REGION Network 14: LH Thermocouple | IW 308
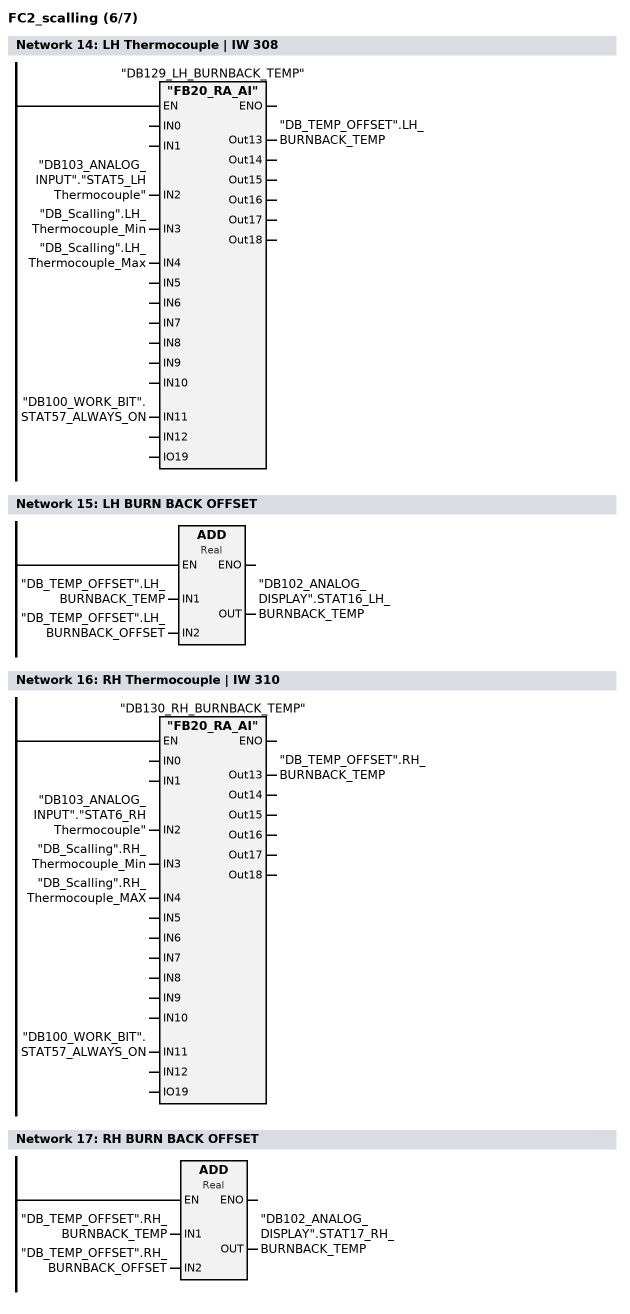
   RUNG wire#powerrail
      "DB129_LH_BURNBACK_TEMP"(IN0 :=, IN1 :=, IN2 := "DB103_ANALOG_INPUT"."STAT5_LH Thermocouple", IN3 := "DB_Scalling".LH_Thermocouple_Min, IN4 := "DB_Scalling".LH_Thermocouple_Max, IN5 :=, IN6 :=, IN7 :=, IN8 :=, IN9 :=, IN10 :=, IN11 := "DB100_WORK_BIT".STAT57_ALWAYS_ON, IN12 :=, IO19 :=, Out13 => "DB_TEMP_OFFSET".LH_BURNBACK_TEMP, Out14 =>, Out15 =>, Out16 =>, Out17 =>, Out18 =>)
   END_RUNG
   // the same network as SCL:
   "DB129_LH_BURNBACK_TEMP"(IN2 := "DB103_ANALOG_INPUT"."STAT5_LH Thermocouple",   // "FB20_RA_AI"
                           IN3 := "DB_Scalling".LH_Thermocouple_Min,
                           IN4 := "DB_Scalling".LH_Thermocouple_Max,
                           IN11 := "DB100_WORK_BIT".STAT57_ALWAYS_ON,
                           Out13 => "DB_TEMP_OFFSET".LH_BURNBACK_TEMP);
END_REGION

REGION Network 15: LH BURN BACK OFFSET
   RUNG wire#powerrail
      { S7_Templates := "SrcType := Real" } Add(in1 := "DB_TEMP_OFFSET".LH_BURNBACK_TEMP, in2 := "DB_TEMP_OFFSET".LH_BURNBACK_OFFSET, out => "DB102_ANALOG_DISPLAY".STAT16_LH_BURNBACK_TEMP)
   END_RUNG
   // the same network as SCL:
   "DB102_ANALOG_DISPLAY".STAT16_LH_BURNBACK_TEMP := "DB_TEMP_OFFSET".LH_BURNBACK_TEMP + "DB_TEMP_OFFSET".LH_BURNBACK_OFFSET;
END_REGION

REGION Network 16: RH Thermocouple | IW 310
   RUNG wire#powerrail
      "DB130_RH_BURNBACK_TEMP"(IN0 :=, IN1 :=, IN2 := "DB103_ANALOG_INPUT"."STAT6_RH Thermocouple", IN3 := "DB_Scalling".RH_Thermocouple_Min, IN4 := "DB_Scalling".RH_Thermocouple_MAX, IN5 :=, IN6 :=, IN7 :=, IN8 :=, IN9 :=, IN10 :=, IN11 := "DB100_WORK_BIT".STAT57_ALWAYS_ON, IN12 :=, IO19 :=, Out13 => "DB_TEMP_OFFSET".RH_BURNBACK_TEMP, Out14 =>, Out15 =>, Out16 =>, Out17 =>, Out18 =>)
   END_RUNG
   // the same network as SCL:
   "DB130_RH_BURNBACK_TEMP"(IN2 := "DB103_ANALOG_INPUT"."STAT6_RH Thermocouple",   // "FB20_RA_AI"
                           IN3 := "DB_Scalling".RH_Thermocouple_Min,
                           IN4 := "DB_Scalling".RH_Thermocouple_MAX,
                           IN11 := "DB100_WORK_BIT".STAT57_ALWAYS_ON,
                           Out13 => "DB_TEMP_OFFSET".RH_BURNBACK_TEMP);
END_REGION

REGION Network 17: RH BURN BACK OFFSET
   RUNG wire#powerrail
      { S7_Templates := "SrcType := Real" } Add(in1 := "DB_TEMP_OFFSET".RH_BURNBACK_TEMP, in2 := "DB_TEMP_OFFSET".RH_BURNBACK_OFFSET, out => "DB102_ANALOG_DISPLAY".STAT17_RH_BURNBACK_TEMP)
   END_RUNG
   // the same network as SCL:
   "DB102_ANALOG_DISPLAY".STAT17_RH_BURNBACK_TEMP := "DB_TEMP_OFFSET".RH_BURNBACK_TEMP + "DB_TEMP_OFFSET".RH_BURNBACK_OFFSET;
END_REGION

REGION Network 18: Poti LH Rear Undgrt | IW 304
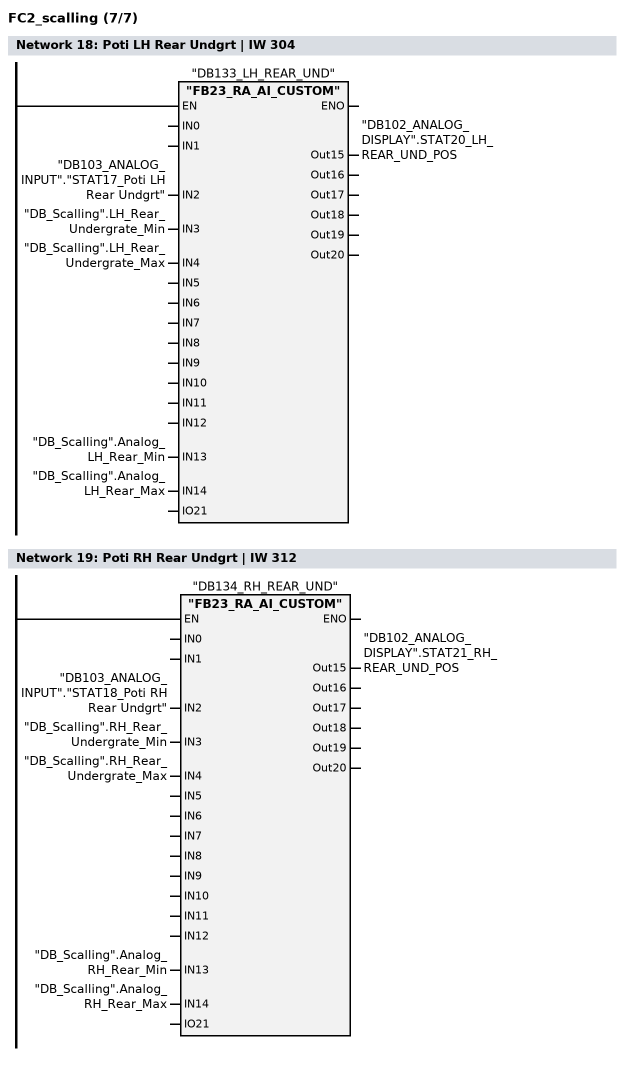
   RUNG wire#powerrail
      "DB133_LH_REAR_UND"(IN0 :=, IN1 :=, IN2 := "DB103_ANALOG_INPUT"."STAT17_Poti LH Rear Undgrt", IN3 := "DB_Scalling".LH_Rear_Undergrate_Min, IN4 := "DB_Scalling".LH_Rear_Undergrate_Max, IN5 :=, IN6 :=, IN7 :=, IN8 :=, IN9 :=, IN10 :=, IN11 :=, IN12 :=, IN13 := "DB_Scalling".Analog_LH_Rear_Min, IN14 := "DB_Scalling".Analog_LH_Rear_Max, IO21 :=, Out15 => "DB102_ANALOG_DISPLAY".STAT20_LH_REAR_UND_POS, Out16 =>, Out17 =>, Out18 =>, Out19 =>, Out20 =>)
   END_RUNG
   // the same network as SCL:
   "DB133_LH_REAR_UND"(IN2 := "DB103_ANALOG_INPUT"."STAT17_Poti LH Rear Undgrt",   // "FB23_RA_AI_CUSTOM"
                       IN3 := "DB_Scalling".LH_Rear_Undergrate_Min,
                       IN4 := "DB_Scalling".LH_Rear_Undergrate_Max,
                       IN13 := "DB_Scalling".Analog_LH_Rear_Min,
                       IN14 := "DB_Scalling".Analog_LH_Rear_Max,
                       Out15 => "DB102_ANALOG_DISPLAY".STAT20_LH_REAR_UND_POS);
END_REGION

REGION Network 19: Poti RH Rear Undgrt | IW 312
   RUNG wire#powerrail
      "DB134_RH_REAR_UND"(IN0 :=, IN1 :=, IN2 := "DB103_ANALOG_INPUT"."STAT18_Poti RH Rear Undgrt", IN3 := "DB_Scalling".RH_Rear_Undergrate_Min, IN4 := "DB_Scalling".RH_Rear_Undergrate_Max, IN5 :=, IN6 :=, IN7 :=, IN8 :=, IN9 :=, IN10 :=, IN11 :=, IN12 :=, IN13 := "DB_Scalling".Analog_RH_Rear_Min, IN14 := "DB_Scalling".Analog_RH_Rear_Max, IO21 :=, Out15 => "DB102_ANALOG_DISPLAY".STAT21_RH_REAR_UND_POS, Out16 =>, Out17 =>, Out18 =>, Out19 =>, Out20 =>)
   END_RUNG
   // the same network as SCL:
   "DB134_RH_REAR_UND"(IN2 := "DB103_ANALOG_INPUT"."STAT18_Poti RH Rear Undgrt",   // "FB23_RA_AI_CUSTOM"
                       IN3 := "DB_Scalling".RH_Rear_Undergrate_Min,
                       IN4 := "DB_Scalling".RH_Rear_Undergrate_Max,
                       IN13 := "DB_Scalling".Analog_RH_Rear_Min,
                       IN14 := "DB_Scalling".Analog_RH_Rear_Max,
                       Out15 => "DB102_ANALOG_DISPLAY".STAT21_RH_REAR_UND_POS);
END_REGION
END_FUNCTION

FUNCTION "FC3_BOILER_OPERATION" : Void   // FC3, LAD
TITLE = BOILER OPERATION
{ S7_Optimized_Access := 'TRUE' }
VERSION : 0.1
BEGIN

REGION Network 1: Ready For Operation ==> I 0.1
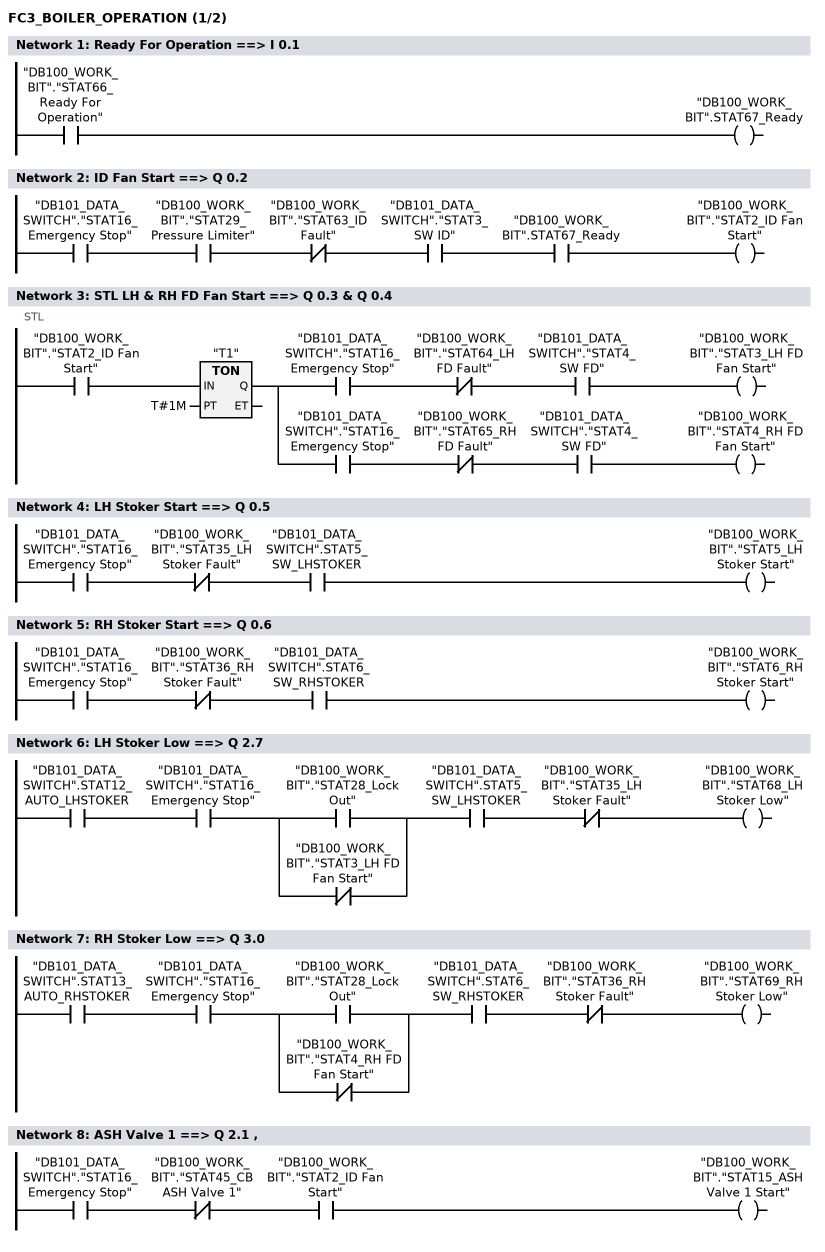
   RUNG wire#powerrail
      Contact( "DB100_WORK_BIT"."STAT66_Ready For Operation" )
      Coil( "DB100_WORK_BIT".STAT67_Ready )
   END_RUNG
   // the same network as SCL:
   "DB100_WORK_BIT".STAT67_Ready := "DB100_WORK_BIT"."STAT66_Ready For Operation";
END_REGION

REGION Network 2: ID Fan Start ==> Q 0.2
   RUNG wire#powerrail
      Contact( "DB101_DATA_SWITCH"."STAT16_Emergency Stop" )
      Contact( "DB100_WORK_BIT"."STAT29_Pressure Limiter" )
      I_Contact( "DB100_WORK_BIT"."STAT63_ID Fault" )
      Contact( "DB101_DATA_SWITCH"."STAT3_SW ID" )
      Contact( "DB100_WORK_BIT".STAT67_Ready )
      Coil( "DB100_WORK_BIT"."STAT2_ID Fan Start" )
   END_RUNG
   // the same network as SCL:
   "DB100_WORK_BIT"."STAT2_ID Fan Start" := "DB101_DATA_SWITCH"."STAT16_Emergency Stop" AND "DB100_WORK_BIT"."STAT29_Pressure Limiter" AND NOT "DB100_WORK_BIT"."STAT63_ID Fault" AND "DB101_DATA_SWITCH"."STAT3_SW ID" AND "DB100_WORK_BIT".STAT67_Ready;
END_REGION

REGION Network 3: STL LH & RH FD Fan Start ==> Q 0.3 & Q 0.4
   // STL
   "T1".TON(IN := "DB100_WORK_BIT"."STAT2_ID Fan Start", PT := T#1M);
   "DB100_WORK_BIT"."STAT3_LH FD Fan Start" := "T1".Q AND "DB101_DATA_SWITCH"."STAT16_Emergency Stop" AND NOT "DB100_WORK_BIT"."STAT64_LH FD Fault" AND "DB101_DATA_SWITCH"."STAT4_SW FD";
   "DB100_WORK_BIT"."STAT4_RH FD Fan Start" := "T1".Q AND "DB101_DATA_SWITCH"."STAT16_Emergency Stop" AND NOT "DB100_WORK_BIT"."STAT65_RH FD Fault" AND "DB101_DATA_SWITCH"."STAT4_SW FD";
END_REGION

REGION Network 4: LH Stoker Start ==> Q 0.5
   RUNG wire#powerrail
      Contact( "DB101_DATA_SWITCH"."STAT16_Emergency Stop" )
      I_Contact( "DB100_WORK_BIT"."STAT35_LH Stoker Fault" )
      Contact( "DB101_DATA_SWITCH".STAT5_SW_LHSTOKER )
      Coil( "DB100_WORK_BIT"."STAT5_LH Stoker Start" )
   END_RUNG
   // the same network as SCL:
   "DB100_WORK_BIT"."STAT5_LH Stoker Start" := "DB101_DATA_SWITCH"."STAT16_Emergency Stop" AND NOT "DB100_WORK_BIT"."STAT35_LH Stoker Fault" AND "DB101_DATA_SWITCH".STAT5_SW_LHSTOKER;
END_REGION

REGION Network 5: RH Stoker Start ==> Q 0.6
   RUNG wire#powerrail
      Contact( "DB101_DATA_SWITCH"."STAT16_Emergency Stop" )
      I_Contact( "DB100_WORK_BIT"."STAT36_RH Stoker Fault" )
      Contact( "DB101_DATA_SWITCH".STAT6_SW_RHSTOKER )
      Coil( "DB100_WORK_BIT"."STAT6_RH Stoker Start" )
   END_RUNG
   // the same network as SCL:
   "DB100_WORK_BIT"."STAT6_RH Stoker Start" := "DB101_DATA_SWITCH"."STAT16_Emergency Stop" AND NOT "DB100_WORK_BIT"."STAT36_RH Stoker Fault" AND "DB101_DATA_SWITCH".STAT6_SW_RHSTOKER;
END_REGION

REGION Network 6: LH Stoker Low ==> Q 2.7
   RUNG wire#powerrail
      Contact( "DB101_DATA_SWITCH".STAT12_AUTO_LHSTOKER )
      Contact( "DB101_DATA_SWITCH"."STAT16_Emergency Stop" )
      wire#w1
      Contact( "DB100_WORK_BIT"."STAT28_Lock Out" )
      wire#w2
      Contact( "DB101_DATA_SWITCH".STAT5_SW_LHSTOKER )
      I_Contact( "DB100_WORK_BIT"."STAT35_LH Stoker Fault" )
      Coil( "DB100_WORK_BIT"."STAT68_LH Stoker Low" )
   END_RUNG
   RUNG wire#w1
      I_Contact( "DB100_WORK_BIT"."STAT3_LH FD Fan Start" )
   END_RUNG wire#w2
   // the same network as SCL:
   "DB100_WORK_BIT"."STAT68_LH Stoker Low" := "DB101_DATA_SWITCH".STAT12_AUTO_LHSTOKER AND "DB101_DATA_SWITCH"."STAT16_Emergency Stop" AND ("DB100_WORK_BIT"."STAT28_Lock Out" OR NOT "DB100_WORK_BIT"."STAT3_LH FD Fan Start") AND "DB101_DATA_SWITCH".STAT5_SW_LHSTOKER AND NOT "DB100_WORK_BIT"."STAT35_LH Stoker Fault";
END_REGION

REGION Network 7: RH Stoker Low ==> Q 3.0
   RUNG wire#powerrail
      Contact( "DB101_DATA_SWITCH".STAT13_AUTO_RHSTOKER )
      Contact( "DB101_DATA_SWITCH"."STAT16_Emergency Stop" )
      wire#w1
      Contact( "DB100_WORK_BIT"."STAT28_Lock Out" )
      wire#w2
      Contact( "DB101_DATA_SWITCH".STAT6_SW_RHSTOKER )
      I_Contact( "DB100_WORK_BIT"."STAT36_RH Stoker Fault" )
      Coil( "DB100_WORK_BIT"."STAT69_RH Stoker Low" )
   END_RUNG
   RUNG wire#w1
      I_Contact( "DB100_WORK_BIT"."STAT4_RH FD Fan Start" )
   END_RUNG wire#w2
   // the same network as SCL:
   "DB100_WORK_BIT"."STAT69_RH Stoker Low" := "DB101_DATA_SWITCH".STAT13_AUTO_RHSTOKER AND "DB101_DATA_SWITCH"."STAT16_Emergency Stop" AND ("DB100_WORK_BIT"."STAT28_Lock Out" OR NOT "DB100_WORK_BIT"."STAT4_RH FD Fan Start") AND "DB101_DATA_SWITCH".STAT6_SW_RHSTOKER AND NOT "DB100_WORK_BIT"."STAT36_RH Stoker Fault";
END_REGION

REGION Network 8: ASH Valve 1 ==> Q 2.1 ,
   RUNG wire#powerrail
      Contact( "DB101_DATA_SWITCH"."STAT16_Emergency Stop" )
      I_Contact( "DB100_WORK_BIT"."STAT45_CB ASH Valve 1" )
      Contact( "DB100_WORK_BIT"."STAT2_ID Fan Start" )
      Coil( "DB100_WORK_BIT"."STAT15_ASH Valve 1 Start" )
   END_RUNG
   // the same network as SCL:
   "DB100_WORK_BIT"."STAT15_ASH Valve 1 Start" := "DB101_DATA_SWITCH"."STAT16_Emergency Stop" AND NOT "DB100_WORK_BIT"."STAT45_CB ASH Valve 1" AND "DB100_WORK_BIT"."STAT2_ID Fan Start";
END_REGION

REGION Network 9: ASH Valve 2 ==> Q 2.2
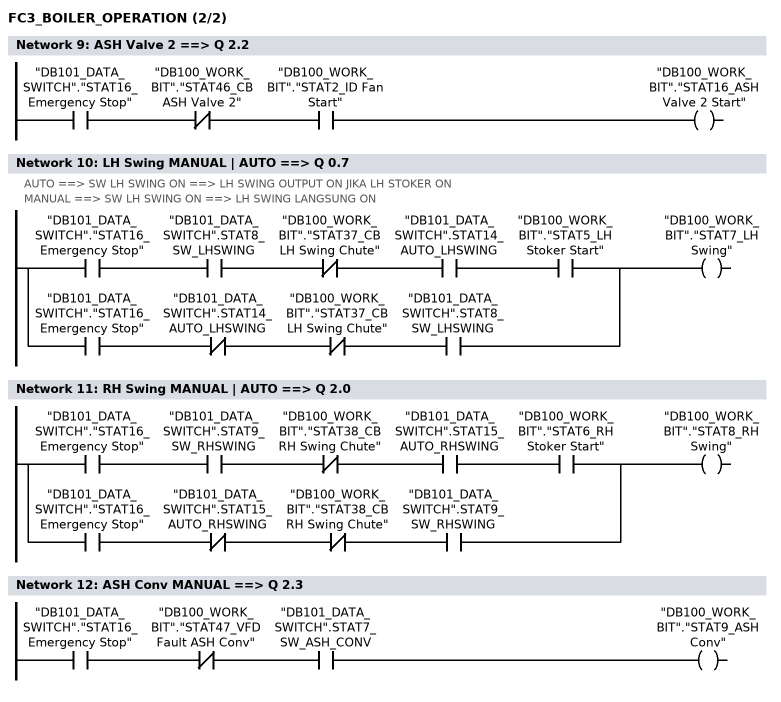
   RUNG wire#powerrail
      Contact( "DB101_DATA_SWITCH"."STAT16_Emergency Stop" )
      I_Contact( "DB100_WORK_BIT"."STAT46_CB ASH Valve 2" )
      Contact( "DB100_WORK_BIT"."STAT2_ID Fan Start" )
      Coil( "DB100_WORK_BIT"."STAT16_ASH Valve 2 Start" )
   END_RUNG
   // the same network as SCL:
   "DB100_WORK_BIT"."STAT16_ASH Valve 2 Start" := "DB101_DATA_SWITCH"."STAT16_Emergency Stop" AND NOT "DB100_WORK_BIT"."STAT46_CB ASH Valve 2" AND "DB100_WORK_BIT"."STAT2_ID Fan Start";
END_REGION

REGION Network 10: LH Swing MANUAL | AUTO ==> Q 0.7
   // AUTO ==> SW LH SWING ON ==> LH SWING OUTPUT ON JIKA LH STOKER ON
   // MANUAL ==> SW LH SWING ON ==> LH SWING LANGSUNG ON
   RUNG wire#powerrail
      Contact( "DB101_DATA_SWITCH"."STAT16_Emergency Stop" )
      Contact( "DB101_DATA_SWITCH".STAT8_SW_LHSWING )
      I_Contact( "DB100_WORK_BIT"."STAT37_CB LH Swing Chute" )
      Contact( "DB101_DATA_SWITCH".STAT14_AUTO_LHSWING )
      Contact( "DB100_WORK_BIT"."STAT5_LH Stoker Start" )
      wire#w1
      Coil( "DB100_WORK_BIT"."STAT7_LH Swing" )
   END_RUNG
   RUNG wire#powerrail
      Contact( "DB101_DATA_SWITCH"."STAT16_Emergency Stop" )
      I_Contact( "DB101_DATA_SWITCH".STAT14_AUTO_LHSWING )
      I_Contact( "DB100_WORK_BIT"."STAT37_CB LH Swing Chute" )
      Contact( "DB101_DATA_SWITCH".STAT8_SW_LHSWING )
   END_RUNG wire#w1
   // the same network as SCL:
   "DB100_WORK_BIT"."STAT7_LH Swing" := ("DB101_DATA_SWITCH"."STAT16_Emergency Stop" AND "DB101_DATA_SWITCH".STAT8_SW_LHSWING AND NOT "DB100_WORK_BIT"."STAT37_CB LH Swing Chute" AND "DB101_DATA_SWITCH".STAT14_AUTO_LHSWING AND "DB100_WORK_BIT"."STAT5_LH Stoker Start") OR ("DB101_DATA_SWITCH"."STAT16_Emergency Stop" AND NOT "DB101_DATA_SWITCH".STAT14_AUTO_LHSWING AND NOT "DB100_WORK_BIT"."STAT37_CB LH Swing Chute" AND "DB101_DATA_SWITCH".STAT8_SW_LHSWING);
END_REGION

REGION Network 11: RH Swing MANUAL | AUTO ==> Q 2.0
   RUNG wire#powerrail
      Contact( "DB101_DATA_SWITCH"."STAT16_Emergency Stop" )
      Contact( "DB101_DATA_SWITCH".STAT9_SW_RHSWING )
      I_Contact( "DB100_WORK_BIT"."STAT38_CB RH Swing Chute" )
      Contact( "DB101_DATA_SWITCH".STAT15_AUTO_RHSWING )
      Contact( "DB100_WORK_BIT"."STAT6_RH Stoker Start" )
      wire#w1
      Coil( "DB100_WORK_BIT"."STAT8_RH Swing" )
   END_RUNG
   RUNG wire#powerrail
      Contact( "DB101_DATA_SWITCH"."STAT16_Emergency Stop" )
      I_Contact( "DB101_DATA_SWITCH".STAT15_AUTO_RHSWING )
      I_Contact( "DB100_WORK_BIT"."STAT38_CB RH Swing Chute" )
      Contact( "DB101_DATA_SWITCH".STAT9_SW_RHSWING )
   END_RUNG wire#w1
   // the same network as SCL:
   "DB100_WORK_BIT"."STAT8_RH Swing" := ("DB101_DATA_SWITCH"."STAT16_Emergency Stop" AND "DB101_DATA_SWITCH".STAT9_SW_RHSWING AND NOT "DB100_WORK_BIT"."STAT38_CB RH Swing Chute" AND "DB101_DATA_SWITCH".STAT15_AUTO_RHSWING AND "DB100_WORK_BIT"."STAT6_RH Stoker Start") OR ("DB101_DATA_SWITCH"."STAT16_Emergency Stop" AND NOT "DB101_DATA_SWITCH".STAT15_AUTO_RHSWING AND NOT "DB100_WORK_BIT"."STAT38_CB RH Swing Chute" AND "DB101_DATA_SWITCH".STAT9_SW_RHSWING);
END_REGION

REGION Network 12: ASH Conv MANUAL ==> Q 2.3
   RUNG wire#powerrail
      Contact( "DB101_DATA_SWITCH"."STAT16_Emergency Stop" )
      I_Contact( "DB100_WORK_BIT"."STAT47_VFD Fault ASH Conv" )
      Contact( "DB101_DATA_SWITCH".STAT7_SW_ASH_CONV )
      Coil( "DB100_WORK_BIT"."STAT9_ASH Conv" )
   END_RUNG
   // the same network as SCL:
   "DB100_WORK_BIT"."STAT9_ASH Conv" := "DB101_DATA_SWITCH"."STAT16_Emergency Stop" AND NOT "DB100_WORK_BIT"."STAT47_VFD Fault ASH Conv" AND "DB101_DATA_SWITCH".STAT7_SW_ASH_CONV;
END_REGION
END_FUNCTION

FUNCTION "FC4_ID_SPEED_CONTROL" : Void   // FC4, LAD
TITLE = ID FAN SPEED CONTROL WITH PHOTOHELIC
{ S7_Optimized_Access := 'TRUE' }
VERSION : 0.1
// ID FAN REFF SPEED AO = QW 504
// 
// PHOTOHELIC NO = I 4.6
// PHOTOHELIC NC = I 4.7
BEGIN

REGION Network 1: ID FAN MODE|AUTO(PHOTOHELIC NC ) | MANUAL(HMI)| SPEED UP
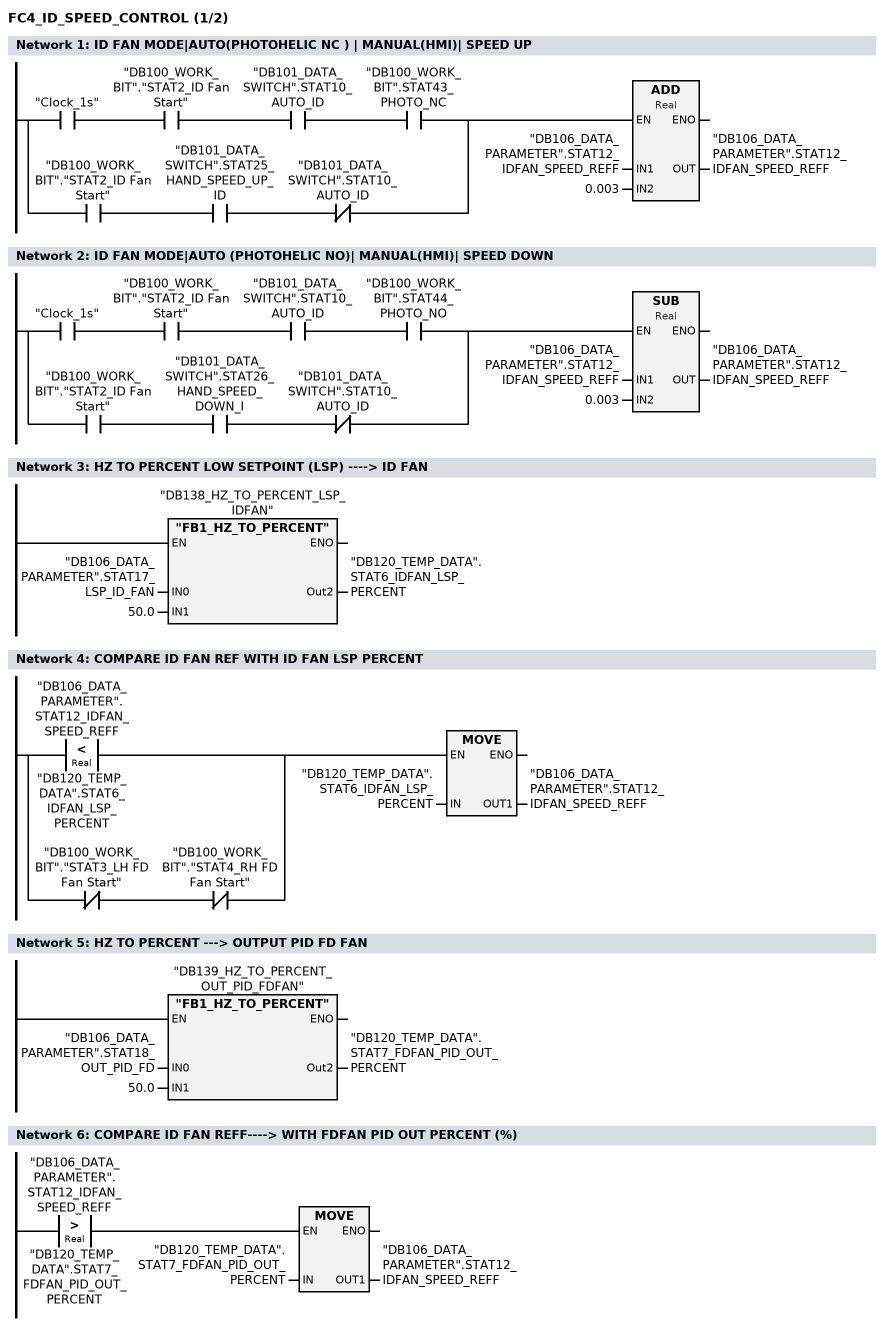
   RUNG wire#powerrail
      Contact( "Clock_1s" )
      Contact( "DB100_WORK_BIT"."STAT2_ID Fan Start" )
      Contact( "DB101_DATA_SWITCH".STAT10_AUTO_ID )
      Contact( "DB100_WORK_BIT".STAT43_PHOTO_NC )
      wire#w1
      { S7_Templates := "SrcType := Real" } Add(in1 := "DB106_DATA_PARAMETER".STAT12_IDFAN_SPEED_REFF, in2 := 0.003, out => "DB106_DATA_PARAMETER".STAT12_IDFAN_SPEED_REFF)
   END_RUNG
   RUNG wire#powerrail
      Contact( "DB100_WORK_BIT"."STAT2_ID Fan Start" )
      Contact( "DB101_DATA_SWITCH".STAT25_HAND_SPEED_UP_ID )
      I_Contact( "DB101_DATA_SWITCH".STAT10_AUTO_ID )
   END_RUNG wire#w1
   // the same network as SCL:
   IF ("Clock_1s" AND "DB100_WORK_BIT"."STAT2_ID Fan Start" AND "DB101_DATA_SWITCH".STAT10_AUTO_ID AND "DB100_WORK_BIT".STAT43_PHOTO_NC) OR ("DB100_WORK_BIT"."STAT2_ID Fan Start" AND "DB101_DATA_SWITCH".STAT25_HAND_SPEED_UP_ID AND NOT "DB101_DATA_SWITCH".STAT10_AUTO_ID) THEN
       "DB106_DATA_PARAMETER".STAT12_IDFAN_SPEED_REFF := "DB106_DATA_PARAMETER".STAT12_IDFAN_SPEED_REFF + 0.003;
   END_IF;
END_REGION

REGION Network 2: ID FAN MODE|AUTO (PHOTOHELIC NO)| MANUAL(HMI)| SPEED DOWN
   RUNG wire#powerrail
      Contact( "Clock_1s" )
      Contact( "DB100_WORK_BIT"."STAT2_ID Fan Start" )
      Contact( "DB101_DATA_SWITCH".STAT10_AUTO_ID )
      Contact( "DB100_WORK_BIT".STAT44_PHOTO_NO )
      wire#w1
      { S7_Templates := "SrcType := Real" } Sub(in1 := "DB106_DATA_PARAMETER".STAT12_IDFAN_SPEED_REFF, in2 := 0.003, out => "DB106_DATA_PARAMETER".STAT12_IDFAN_SPEED_REFF)
   END_RUNG
   RUNG wire#powerrail
      Contact( "DB100_WORK_BIT"."STAT2_ID Fan Start" )
      Contact( "DB101_DATA_SWITCH".STAT26_HAND_SPEED_DOWN_I )
      I_Contact( "DB101_DATA_SWITCH".STAT10_AUTO_ID )
   END_RUNG wire#w1
   // the same network as SCL:
   IF ("Clock_1s" AND "DB100_WORK_BIT"."STAT2_ID Fan Start" AND "DB101_DATA_SWITCH".STAT10_AUTO_ID AND "DB100_WORK_BIT".STAT44_PHOTO_NO) OR ("DB100_WORK_BIT"."STAT2_ID Fan Start" AND "DB101_DATA_SWITCH".STAT26_HAND_SPEED_DOWN_I AND NOT "DB101_DATA_SWITCH".STAT10_AUTO_ID) THEN
       "DB106_DATA_PARAMETER".STAT12_IDFAN_SPEED_REFF := "DB106_DATA_PARAMETER".STAT12_IDFAN_SPEED_REFF - 0.003;
   END_IF;
END_REGION

REGION Network 3: HZ TO PERCENT LOW SETPOINT (LSP) ----> ID FAN
   RUNG wire#powerrail
      "DB138_HZ_TO_PERCENT_LSP_IDFAN"(IN0 := "DB106_DATA_PARAMETER".STAT17_LSP_ID_FAN, IN1 := 50.0, Out2 => "DB120_TEMP_DATA".STAT6_IDFAN_LSP_PERCENT)
   END_RUNG
   // the same network as SCL:
   "DB138_HZ_TO_PERCENT_LSP_IDFAN"(IN0 := "DB106_DATA_PARAMETER".STAT17_LSP_ID_FAN,   // "FB1_HZ_TO_PERCENT"
                           IN1 := 50.0,
                           Out2 => "DB120_TEMP_DATA".STAT6_IDFAN_LSP_PERCENT);
END_REGION

REGION Network 4: COMPARE ID FAN REF WITH ID FAN LSP PERCENT
   RUNG wire#powerrail
      { S7_Templates := "SrcType := Real" } LT_Contact(in1 := "DB106_DATA_PARAMETER".STAT12_IDFAN_SPEED_REFF, in2 := "DB120_TEMP_DATA".STAT6_IDFAN_LSP_PERCENT)
      wire#w1
      Move(in := "DB120_TEMP_DATA".STAT6_IDFAN_LSP_PERCENT, out1 => "DB106_DATA_PARAMETER".STAT12_IDFAN_SPEED_REFF)
   END_RUNG
   RUNG wire#powerrail
      I_Contact( "DB100_WORK_BIT"."STAT3_LH FD Fan Start" )
      I_Contact( "DB100_WORK_BIT"."STAT4_RH FD Fan Start" )
   END_RUNG wire#w1
   // the same network as SCL:
   IF ("DB106_DATA_PARAMETER".STAT12_IDFAN_SPEED_REFF < "DB120_TEMP_DATA".STAT6_IDFAN_LSP_PERCENT) OR (NOT "DB100_WORK_BIT"."STAT3_LH FD Fan Start" AND NOT "DB100_WORK_BIT"."STAT4_RH FD Fan Start") THEN
       "DB106_DATA_PARAMETER".STAT12_IDFAN_SPEED_REFF := "DB120_TEMP_DATA".STAT6_IDFAN_LSP_PERCENT;
   END_IF;
END_REGION

REGION Network 5: HZ TO PERCENT ---> OUTPUT PID FD FAN
   RUNG wire#powerrail
      "DB139_HZ_TO_PERCENT_OUT_PID_FDFAN"(IN0 := "DB106_DATA_PARAMETER".STAT18_OUT_PID_FD, IN1 := 50.0, Out2 => "DB120_TEMP_DATA".STAT7_FDFAN_PID_OUT_PERCENT)
   END_RUNG
   // the same network as SCL:
   "DB139_HZ_TO_PERCENT_OUT_PID_FDFAN"(IN0 := "DB106_DATA_PARAMETER".STAT18_OUT_PID_FD,   // "FB1_HZ_TO_PERCENT"
                           IN1 := 50.0,
                           Out2 => "DB120_TEMP_DATA".STAT7_FDFAN_PID_OUT_PERCENT);
END_REGION

REGION Network 6: COMPARE ID FAN REFF----> WITH FDFAN PID OUT PERCENT (%)
   RUNG wire#powerrail
      { S7_Templates := "SrcType := Real" } GT_Contact(in1 := "DB106_DATA_PARAMETER".STAT12_IDFAN_SPEED_REFF, in2 := "DB120_TEMP_DATA".STAT7_FDFAN_PID_OUT_PERCENT)
      Move(in := "DB120_TEMP_DATA".STAT7_FDFAN_PID_OUT_PERCENT, out1 => "DB106_DATA_PARAMETER".STAT12_IDFAN_SPEED_REFF)
   END_RUNG
   // the same network as SCL:
   IF "DB106_DATA_PARAMETER".STAT12_IDFAN_SPEED_REFF > "DB120_TEMP_DATA".STAT7_FDFAN_PID_OUT_PERCENT THEN
       "DB106_DATA_PARAMETER".STAT12_IDFAN_SPEED_REFF := "DB120_TEMP_DATA".STAT7_FDFAN_PID_OUT_PERCENT;
   END_IF;
END_REGION

REGION Network 7: {SCALING } ID FAN REFERENCE SPEED AO( QW 504)
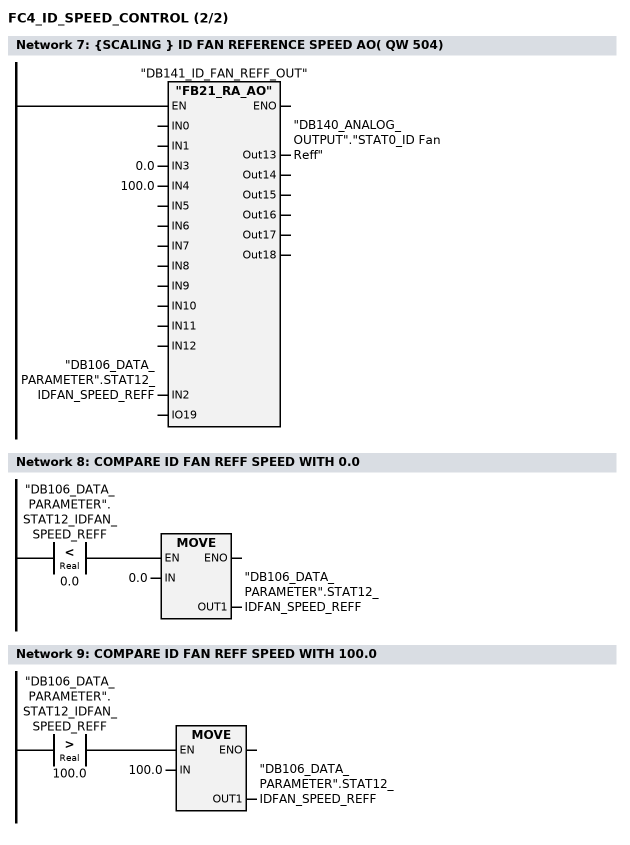
   RUNG wire#powerrail
      "DB141_ID_FAN_REFF_OUT"(IN0 :=, IN1 :=, IN3 := 0.0, IN4 := 100.0, IN5 :=, IN6 :=, IN7 :=, IN8 :=, IN9 :=, IN10 :=, IN11 :=, IN12 :=, IN2 := "DB106_DATA_PARAMETER".STAT12_IDFAN_SPEED_REFF, IO19 :=, Out13 => "DB140_ANALOG_OUTPUT"."STAT0_ID Fan Reff", Out14 =>, Out15 =>, Out16 =>, Out17 =>, Out18 =>)
   END_RUNG
   // the same network as SCL:
   "DB141_ID_FAN_REFF_OUT"(IN3 := 0.0,   // "FB21_RA_AO"
                           IN4 := 100.0,
                           IN2 := "DB106_DATA_PARAMETER".STAT12_IDFAN_SPEED_REFF,
                           Out13 => "DB140_ANALOG_OUTPUT"."STAT0_ID Fan Reff");
END_REGION

REGION Network 8: COMPARE ID FAN REFF SPEED WITH 0.0
   RUNG wire#powerrail
      { S7_Templates := "SrcType := Real" } LT_Contact(in1 := "DB106_DATA_PARAMETER".STAT12_IDFAN_SPEED_REFF, in2 := 0.0)
      Move(in := 0.0, out1 => "DB106_DATA_PARAMETER".STAT12_IDFAN_SPEED_REFF)
   END_RUNG
   // the same network as SCL:
   IF "DB106_DATA_PARAMETER".STAT12_IDFAN_SPEED_REFF < 0.0 THEN
       "DB106_DATA_PARAMETER".STAT12_IDFAN_SPEED_REFF := 0.0;
   END_IF;
END_REGION

REGION Network 9: COMPARE ID FAN REFF SPEED WITH 100.0
   RUNG wire#powerrail
      { S7_Templates := "SrcType := Real" } GT_Contact(in1 := "DB106_DATA_PARAMETER".STAT12_IDFAN_SPEED_REFF, in2 := 100.0)
      Move(in := 100.0, out1 => "DB106_DATA_PARAMETER".STAT12_IDFAN_SPEED_REFF)
   END_RUNG
   // the same network as SCL:
   IF "DB106_DATA_PARAMETER".STAT12_IDFAN_SPEED_REFF > 100.0 THEN
       "DB106_DATA_PARAMETER".STAT12_IDFAN_SPEED_REFF := 100.0;
   END_IF;
END_REGION
END_FUNCTION

FUNCTION "FC5_FD_SPEED_CONTROL" : Void   // FC5, LAD
TITLE = FD SPEED CONTROL , IW 100(PRESSURE TRANSDUCER),QW 506, QW 600
{ S7_Optimized_Access := 'TRUE' }
VERSION : 0.1
// INPUT PID  = IW 100
// AO SPEED LH FD = QW 506
// AO SPEED RH FD = QW 600
// 
// BLOCK LH FD = Q4.0
// BLOCK RH FD = Q 4.1
   VAR_TEMP
      Out1 : DInt;
      Out2 : Real;
      Out3 : DInt;
      Out4 : Real;
   END_VAR
   VAR_TEMP   // added for the SCL form of the ladder/FBD networks
      _w1 : Bool;
      _w2 : Bool;
   END_VAR
BEGIN

REGION Network 1: MOVE PARAMETER PID FROM HMI
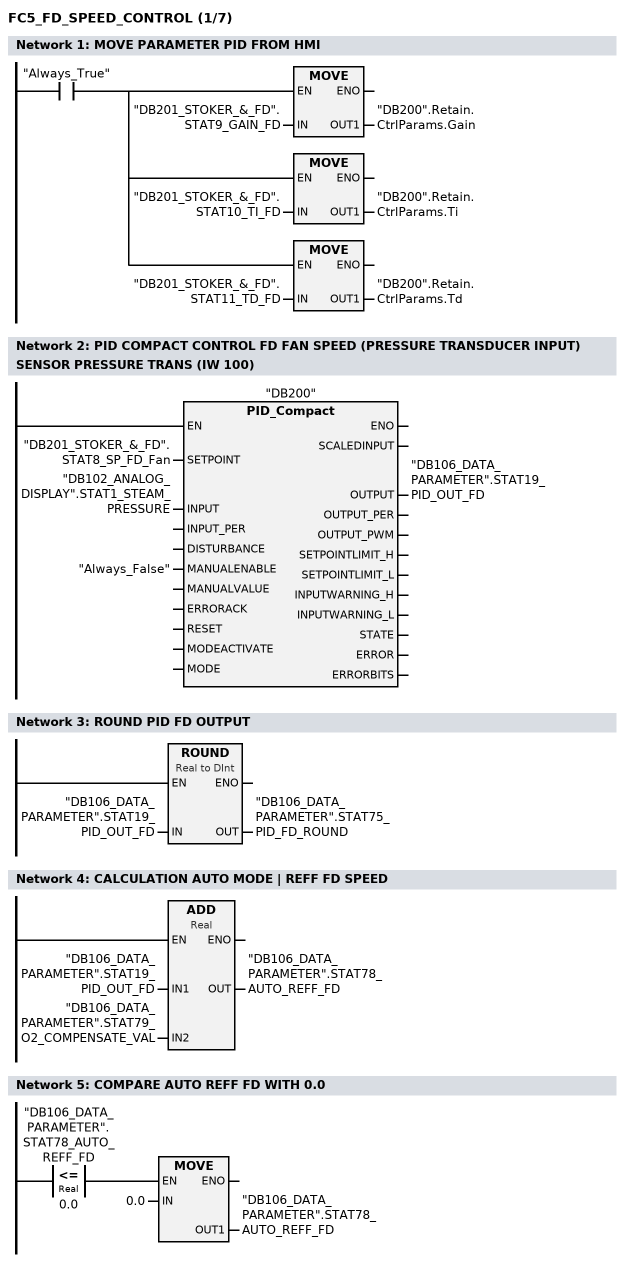
   RUNG wire#powerrail
      Contact( "Always_True" )
      wire#w1
      Move(in := "DB201_STOKER_&_FD".STAT9_GAIN_FD, out1 => "DB200".Retain.CtrlParams.Gain)
   END_RUNG
   RUNG wire#w1
      Move(in := "DB201_STOKER_&_FD".STAT10_TI_FD, out1 => "DB200".Retain.CtrlParams.Ti)
   END_RUNG
   RUNG wire#w1
      Move(in := "DB201_STOKER_&_FD".STAT11_TD_FD, out1 => "DB200".Retain.CtrlParams.Td)
   END_RUNG
   // the same network as SCL:
   IF "Always_True" THEN
       "DB200".Retain.CtrlParams.Gain := "DB201_STOKER_&_FD".STAT9_GAIN_FD;
       "DB200".Retain.CtrlParams.Ti := "DB201_STOKER_&_FD".STAT10_TI_FD;
       "DB200".Retain.CtrlParams.Td := "DB201_STOKER_&_FD".STAT11_TD_FD;
   END_IF;
END_REGION

REGION Network 2: PID COMPACT CONTROL FD FAN SPEED (PRESSURE TRANSDUCER INPUT) SENSOR PRESSURE TRANS (IW 100)
   "DB200"(Setpoint := "DB201_STOKER_&_FD".STAT8_SP_FD_Fan,   // PID_Compact
           Input := "DB102_ANALOG_DISPLAY".STAT1_STEAM_PRESSURE,
           ManualEnable := "Always_False",
           Output => "DB106_DATA_PARAMETER".STAT19_PID_OUT_FD);
END_REGION

REGION Network 3: ROUND PID FD OUTPUT
   RUNG wire#powerrail
      { S7_Templates := "[SrcType := Real, DestType := DInt]" } Round(in := "DB106_DATA_PARAMETER".STAT19_PID_OUT_FD, out => "DB106_DATA_PARAMETER".STAT75_PID_FD_ROUND)
   END_RUNG
   // the same network as SCL:
   "DB106_DATA_PARAMETER".STAT75_PID_FD_ROUND := ROUND("DB106_DATA_PARAMETER".STAT19_PID_OUT_FD);
END_REGION

REGION Network 4: CALCULATION AUTO MODE | REFF FD SPEED
   RUNG wire#powerrail
      { S7_Templates := "SrcType := Real" } Add(in1 := "DB106_DATA_PARAMETER".STAT19_PID_OUT_FD, in2 := "DB106_DATA_PARAMETER".STAT79_O2_COMPENSATE_VAL, out => "DB106_DATA_PARAMETER".STAT78_AUTO_REFF_FD)
   END_RUNG
   // the same network as SCL:
   "DB106_DATA_PARAMETER".STAT78_AUTO_REFF_FD := "DB106_DATA_PARAMETER".STAT19_PID_OUT_FD + "DB106_DATA_PARAMETER".STAT79_O2_COMPENSATE_VAL;
END_REGION

REGION Network 5: COMPARE AUTO REFF FD WITH 0.0
   RUNG wire#powerrail
      { S7_Templates := "SrcType := Real" } LE_Contact(in1 := "DB106_DATA_PARAMETER".STAT78_AUTO_REFF_FD, in2 := 0.0)
      Move(in := 0.0, out1 => "DB106_DATA_PARAMETER".STAT78_AUTO_REFF_FD)
   END_RUNG
   // the same network as SCL:
   IF "DB106_DATA_PARAMETER".STAT78_AUTO_REFF_FD <= 0.0 THEN
       "DB106_DATA_PARAMETER".STAT78_AUTO_REFF_FD := 0.0;
   END_IF;
END_REGION

REGION Network 6: COMPARE AUTO REFF FD WITH 50.0
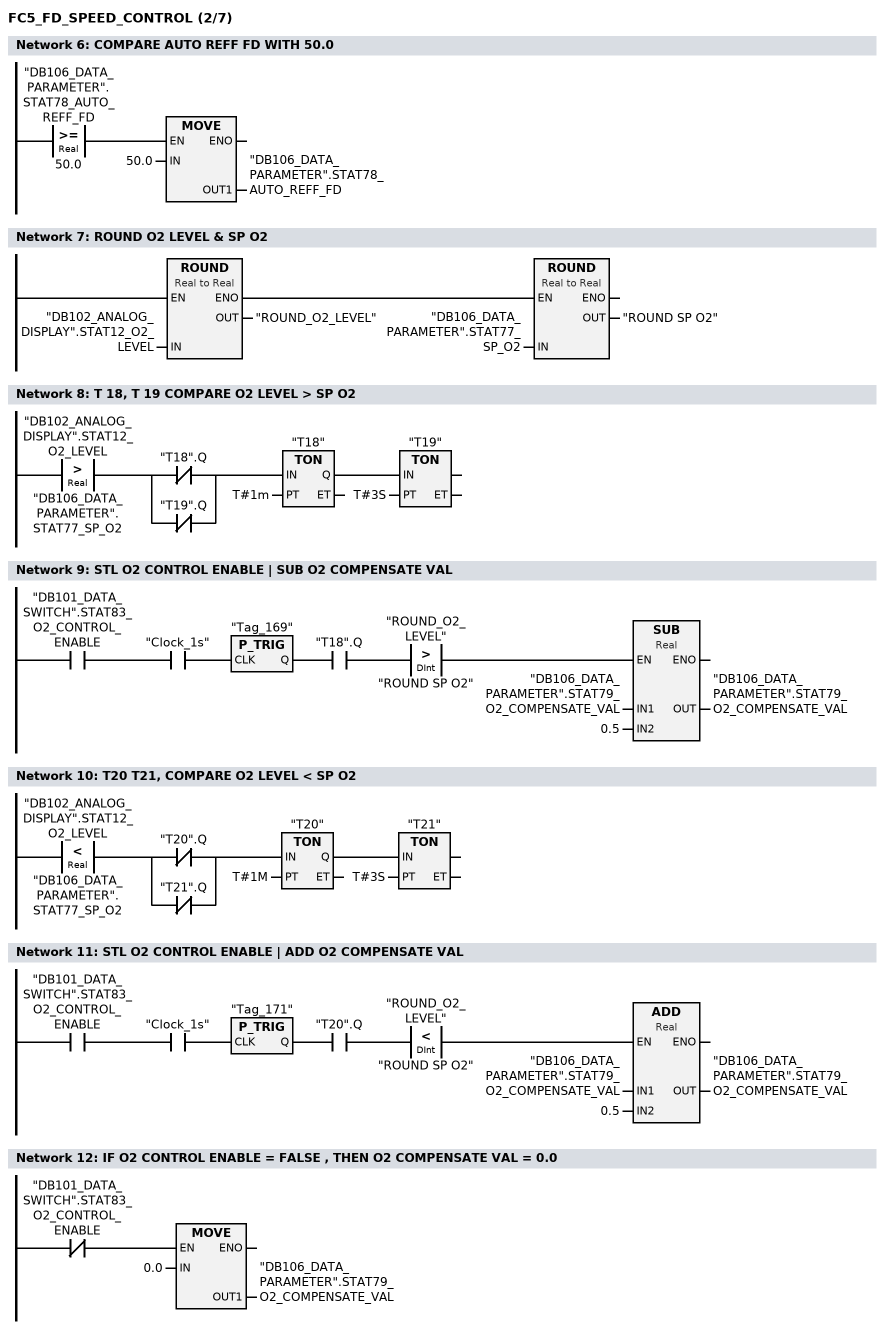
   RUNG wire#powerrail
      { S7_Templates := "SrcType := Real" } GE_Contact(in1 := "DB106_DATA_PARAMETER".STAT78_AUTO_REFF_FD, in2 := 50.0)
      Move(in := 50.0, out1 => "DB106_DATA_PARAMETER".STAT78_AUTO_REFF_FD)
   END_RUNG
   // the same network as SCL:
   IF "DB106_DATA_PARAMETER".STAT78_AUTO_REFF_FD >= 50.0 THEN
       "DB106_DATA_PARAMETER".STAT78_AUTO_REFF_FD := 50.0;
   END_IF;
END_REGION

REGION Network 7: ROUND O2 LEVEL & SP O2
   RUNG wire#powerrail
      { S7_Templates := "[SrcType := Real, DestType := Real]" } Round(in := "DB102_ANALOG_DISPLAY".STAT12_O2_LEVEL, out => "ROUND_O2_LEVEL")
      { S7_Templates := "[SrcType := Real, DestType := Real]" } Round(in := "DB106_DATA_PARAMETER".STAT77_SP_O2, out => "ROUND SP O2")
   END_RUNG
   // the same network as SCL:
   "ROUND_O2_LEVEL" := ROUND("DB102_ANALOG_DISPLAY".STAT12_O2_LEVEL);
   "ROUND SP O2" := ROUND("DB106_DATA_PARAMETER".STAT77_SP_O2);
END_REGION

REGION Network 8: T 18, T 19 COMPARE O2 LEVEL > SP O2
   "T18".TON(IN := ("DB102_ANALOG_DISPLAY".STAT12_O2_LEVEL > "DB106_DATA_PARAMETER".STAT77_SP_O2) AND (NOT "T18".Q OR NOT "T19".Q),
             PT := T#1m);
   "T19".TON(IN := "T18".Q, PT := T#3S);
END_REGION

REGION Network 9: STL O2 CONTROL ENABLE | SUB O2 COMPENSATE VAL
   RUNG wire#powerrail
      Contact( "DB101_DATA_SWITCH".STAT83_O2_CONTROL_ENABLE )
      Contact( "Clock_1s" )
      P_Trig( "Tag_169" )
      Contact( "T18".Q )
      { S7_Templates := "SrcType := DInt" } GT_Contact(in1 := "ROUND_O2_LEVEL", in2 := "ROUND SP O2")
      { S7_Templates := "SrcType := Real" } Sub(in1 := "DB106_DATA_PARAMETER".STAT79_O2_COMPENSATE_VAL, in2 := 0.5, out => "DB106_DATA_PARAMETER".STAT79_O2_COMPENSATE_VAL)
   END_RUNG
   // the same network as SCL:
   #_w1 := "DB101_DATA_SWITCH".STAT83_O2_CONTROL_ENABLE AND "Clock_1s";
   #_w2 := #_w1 AND NOT "Tag_169";   // rising edge
   "Tag_169" := #_w1;
   IF #_w2 AND "T18".Q AND ("ROUND_O2_LEVEL" > "ROUND SP O2") THEN
       "DB106_DATA_PARAMETER".STAT79_O2_COMPENSATE_VAL := "DB106_DATA_PARAMETER".STAT79_O2_COMPENSATE_VAL - 0.5;
   END_IF;
END_REGION

REGION Network 10: T20 T21, COMPARE O2 LEVEL < SP O2
   "T20".TON(IN := ("DB102_ANALOG_DISPLAY".STAT12_O2_LEVEL < "DB106_DATA_PARAMETER".STAT77_SP_O2) AND (NOT "T20".Q OR NOT "T21".Q),
             PT := T#1M);
   "T21".TON(IN := "T20".Q, PT := T#3S);
END_REGION

REGION Network 11: STL O2 CONTROL ENABLE | ADD O2 COMPENSATE VAL
   RUNG wire#powerrail
      Contact( "DB101_DATA_SWITCH".STAT83_O2_CONTROL_ENABLE )
      Contact( "Clock_1s" )
      P_Trig( "Tag_171" )
      Contact( "T20".Q )
      { S7_Templates := "SrcType := DInt" } LT_Contact(in1 := "ROUND_O2_LEVEL", in2 := "ROUND SP O2")
      { S7_Templates := "SrcType := Real" } Add(in1 := "DB106_DATA_PARAMETER".STAT79_O2_COMPENSATE_VAL, in2 := 0.5, out => "DB106_DATA_PARAMETER".STAT79_O2_COMPENSATE_VAL)
   END_RUNG
   // the same network as SCL:
   #_w1 := "DB101_DATA_SWITCH".STAT83_O2_CONTROL_ENABLE AND "Clock_1s";
   #_w2 := #_w1 AND NOT "Tag_171";   // rising edge
   "Tag_171" := #_w1;
   IF #_w2 AND "T20".Q AND ("ROUND_O2_LEVEL" < "ROUND SP O2") THEN
       "DB106_DATA_PARAMETER".STAT79_O2_COMPENSATE_VAL := "DB106_DATA_PARAMETER".STAT79_O2_COMPENSATE_VAL + 0.5;
   END_IF;
END_REGION

REGION Network 12: IF O2 CONTROL ENABLE = FALSE , THEN O2 COMPENSATE VAL = 0.0
   RUNG wire#powerrail
      I_Contact( "DB101_DATA_SWITCH".STAT83_O2_CONTROL_ENABLE )
      Move(in := 0.0, out1 => "DB106_DATA_PARAMETER".STAT79_O2_COMPENSATE_VAL)
   END_RUNG
   // the same network as SCL:
   IF NOT "DB101_DATA_SWITCH".STAT83_O2_CONTROL_ENABLE THEN
       "DB106_DATA_PARAMETER".STAT79_O2_COMPENSATE_VAL := 0.0;
   END_IF;
END_REGION

REGION Network 13: MAXIMUM PERCENT O2
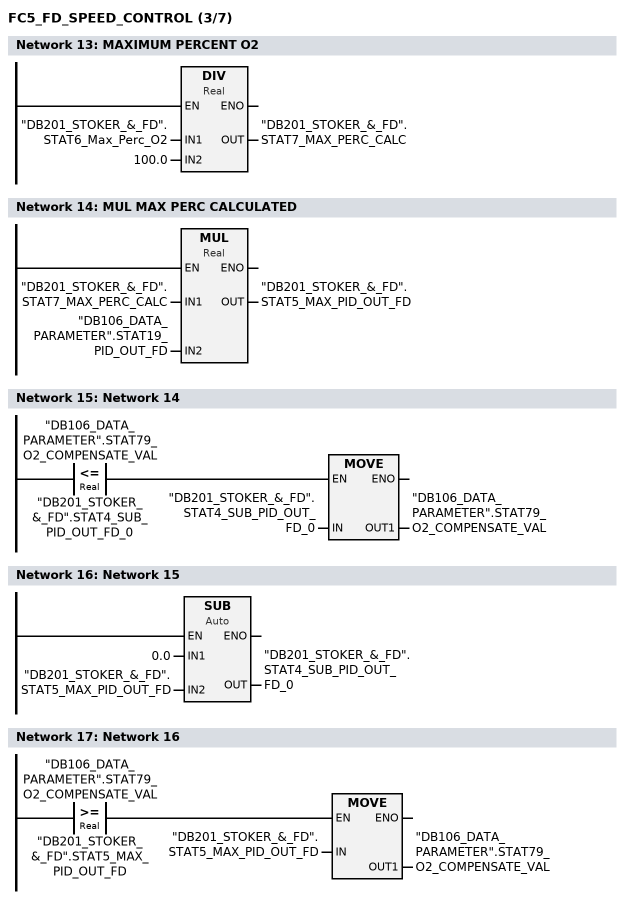
   RUNG wire#powerrail
      { S7_Templates := "SrcType := Real" } Div(in1 := "DB201_STOKER_&_FD".STAT6_Max_Perc_O2, in2 := 100.0, out => "DB201_STOKER_&_FD".STAT7_MAX_PERC_CALC)
   END_RUNG
   // the same network as SCL:
   "DB201_STOKER_&_FD".STAT7_MAX_PERC_CALC := "DB201_STOKER_&_FD".STAT6_Max_Perc_O2 / 100.0;
END_REGION

REGION Network 14: MUL MAX PERC CALCULATED
   RUNG wire#powerrail
      { S7_Templates := "SrcType := Real" } Mul(in1 := "DB201_STOKER_&_FD".STAT7_MAX_PERC_CALC, in2 := "DB106_DATA_PARAMETER".STAT19_PID_OUT_FD, out => "DB201_STOKER_&_FD".STAT5_MAX_PID_OUT_FD)
   END_RUNG
   // the same network as SCL:
   "DB201_STOKER_&_FD".STAT5_MAX_PID_OUT_FD := "DB201_STOKER_&_FD".STAT7_MAX_PERC_CALC * "DB106_DATA_PARAMETER".STAT19_PID_OUT_FD;
END_REGION

REGION Network 15: Network 14
   RUNG wire#powerrail
      { S7_Templates := "SrcType := Real" } LE_Contact(in1 := "DB106_DATA_PARAMETER".STAT79_O2_COMPENSATE_VAL, in2 := "DB201_STOKER_&_FD".STAT4_SUB_PID_OUT_FD_0)
      Move(in := "DB201_STOKER_&_FD".STAT4_SUB_PID_OUT_FD_0, out1 => "DB106_DATA_PARAMETER".STAT79_O2_COMPENSATE_VAL)
   END_RUNG
   // the same network as SCL:
   IF "DB106_DATA_PARAMETER".STAT79_O2_COMPENSATE_VAL <= "DB201_STOKER_&_FD".STAT4_SUB_PID_OUT_FD_0 THEN
       "DB106_DATA_PARAMETER".STAT79_O2_COMPENSATE_VAL := "DB201_STOKER_&_FD".STAT4_SUB_PID_OUT_FD_0;
   END_IF;
END_REGION

REGION Network 16: Network 15
   RUNG wire#powerrail
      Sub(in1 := 0.0, in2 := "DB201_STOKER_&_FD".STAT5_MAX_PID_OUT_FD, out => "DB201_STOKER_&_FD".STAT4_SUB_PID_OUT_FD_0)
   END_RUNG
   // the same network as SCL:
   "DB201_STOKER_&_FD".STAT4_SUB_PID_OUT_FD_0 := 0.0 - "DB201_STOKER_&_FD".STAT5_MAX_PID_OUT_FD;
END_REGION

REGION Network 17: Network 16
   RUNG wire#powerrail
      { S7_Templates := "SrcType := Real" } GE_Contact(in1 := "DB106_DATA_PARAMETER".STAT79_O2_COMPENSATE_VAL, in2 := "DB201_STOKER_&_FD".STAT5_MAX_PID_OUT_FD)
      Move(in := "DB201_STOKER_&_FD".STAT5_MAX_PID_OUT_FD, out1 => "DB106_DATA_PARAMETER".STAT79_O2_COMPENSATE_VAL)
   END_RUNG
   // the same network as SCL:
   IF "DB106_DATA_PARAMETER".STAT79_O2_COMPENSATE_VAL >= "DB201_STOKER_&_FD".STAT5_MAX_PID_OUT_FD THEN
       "DB106_DATA_PARAMETER".STAT79_O2_COMPENSATE_VAL := "DB201_STOKER_&_FD".STAT5_MAX_PID_OUT_FD;
   END_IF;
END_REGION

REGION Network 18: SCALING SPEED REFERENCE LH FD | AUTO | ANALOG OUTPUT (QW 506)
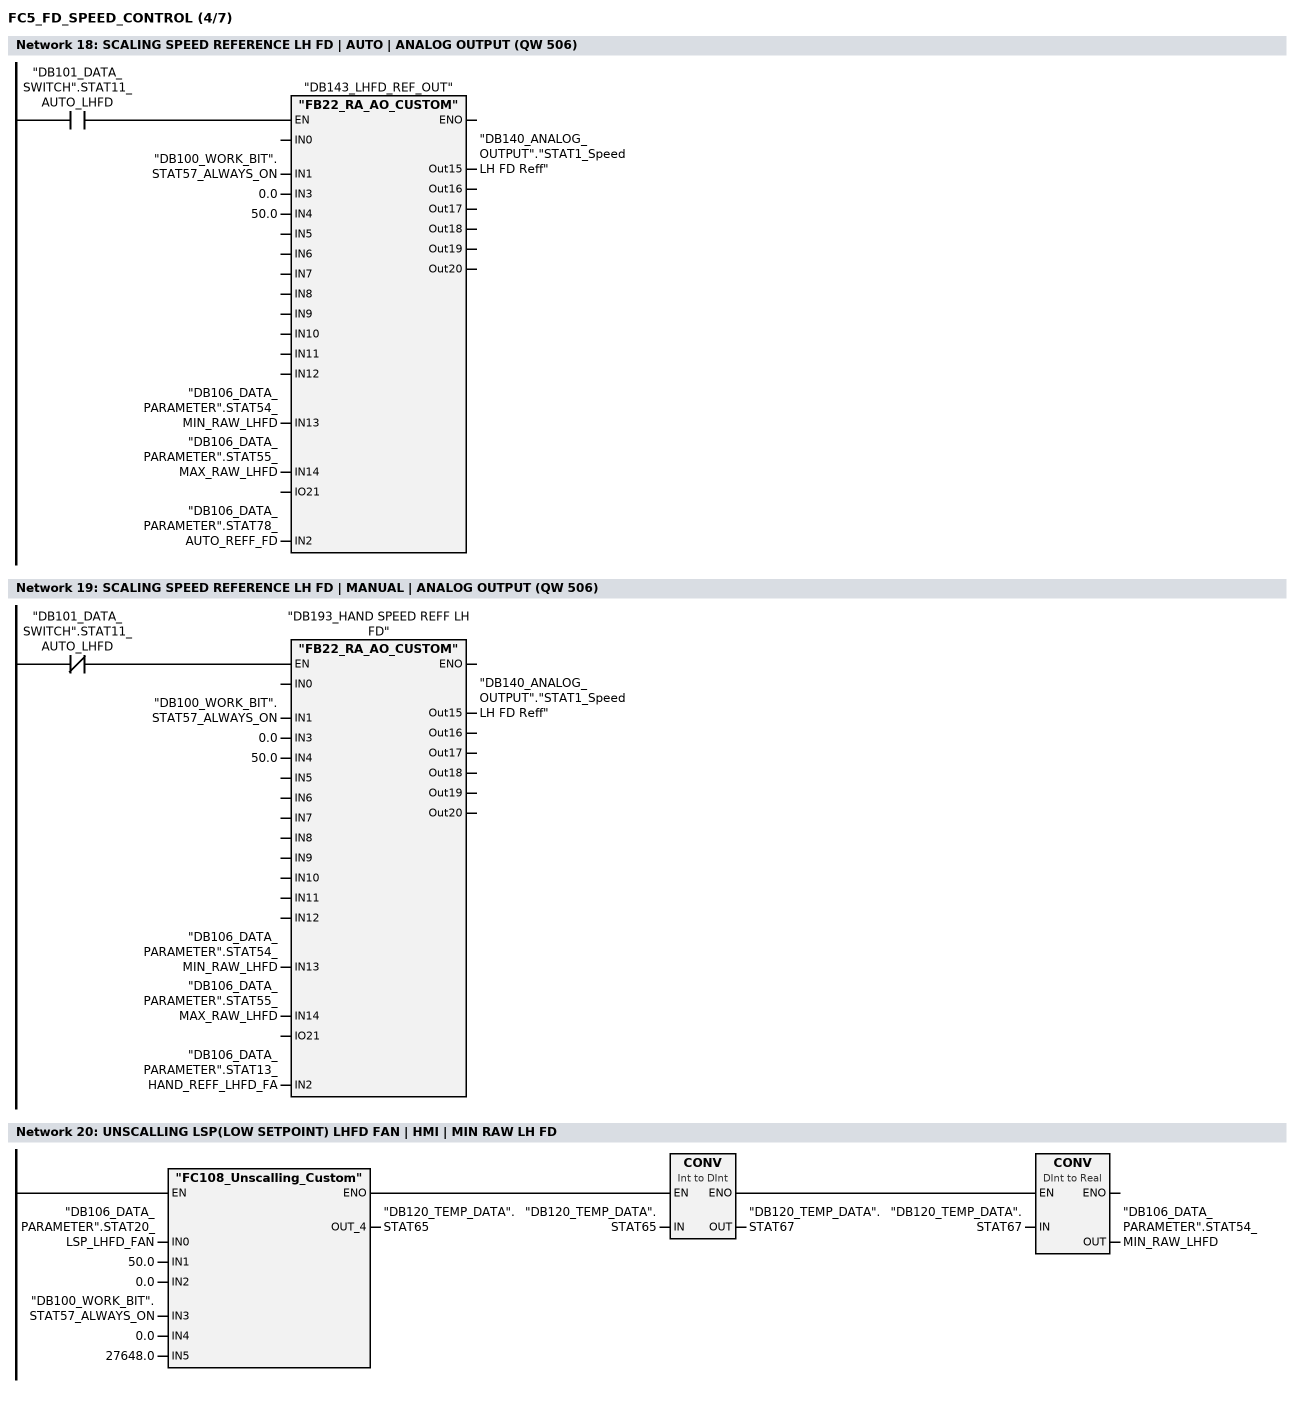
   RUNG wire#powerrail
      Contact( "DB101_DATA_SWITCH".STAT11_AUTO_LHFD )
      "DB143_LHFD_REF_OUT"(IN0 :=, IN1 := "DB100_WORK_BIT".STAT57_ALWAYS_ON, IN3 := 0.0, IN4 := 50.0, IN5 :=, IN6 :=, IN7 :=, IN8 :=, IN9 :=, IN10 :=, IN11 :=, IN12 :=, IN13 := "DB106_DATA_PARAMETER".STAT54_MIN_RAW_LHFD, IN14 := "DB106_DATA_PARAMETER".STAT55_MAX_RAW_LHFD, IO21 :=, IN2 := "DB106_DATA_PARAMETER".STAT78_AUTO_REFF_FD, Out15 => "DB140_ANALOG_OUTPUT"."STAT1_Speed LH FD Reff", Out16 =>, Out17 =>, Out18 =>, Out19 =>, Out20 =>)
   END_RUNG
   // the same network as SCL:
   IF "DB101_DATA_SWITCH".STAT11_AUTO_LHFD THEN
       "DB143_LHFD_REF_OUT"(IN1 := "DB100_WORK_BIT".STAT57_ALWAYS_ON,   // "FB22_RA_AO_CUSTOM"
                            IN3 := 0.0,
                            IN4 := 50.0,
                            IN13 := "DB106_DATA_PARAMETER".STAT54_MIN_RAW_LHFD,
                            IN14 := "DB106_DATA_PARAMETER".STAT55_MAX_RAW_LHFD,
                            IN2 := "DB106_DATA_PARAMETER".STAT78_AUTO_REFF_FD,
                            Out15 => "DB140_ANALOG_OUTPUT"."STAT1_Speed LH FD Reff");
   END_IF;
END_REGION

REGION Network 19: SCALING SPEED REFERENCE LH FD | MANUAL | ANALOG OUTPUT (QW 506)
   RUNG wire#powerrail
      I_Contact( "DB101_DATA_SWITCH".STAT11_AUTO_LHFD )
      "DB193_HAND SPEED REFF LH FD"(IN0 :=, IN1 := "DB100_WORK_BIT".STAT57_ALWAYS_ON, IN3 := 0.0, IN4 := 50.0, IN5 :=, IN6 :=, IN7 :=, IN8 :=, IN9 :=, IN10 :=, IN11 :=, IN12 :=, IN13 := "DB106_DATA_PARAMETER".STAT54_MIN_RAW_LHFD, IN14 := "DB106_DATA_PARAMETER".STAT55_MAX_RAW_LHFD, IO21 :=, IN2 := "DB106_DATA_PARAMETER".STAT13_HAND_REFF_LHFD_FA, Out15 => "DB140_ANALOG_OUTPUT"."STAT1_Speed LH FD Reff", Out16 =>, Out17 =>, Out18 =>, Out19 =>, Out20 =>)
   END_RUNG
   // the same network as SCL:
   IF NOT "DB101_DATA_SWITCH".STAT11_AUTO_LHFD THEN
       "DB193_HAND SPEED REFF LH FD"(IN1 := "DB100_WORK_BIT".STAT57_ALWAYS_ON,   // "FB22_RA_AO_CUSTOM"
                               IN3 := 0.0,
                               IN4 := 50.0,
                               IN13 := "DB106_DATA_PARAMETER".STAT54_MIN_RAW_LHFD,
                               IN14 := "DB106_DATA_PARAMETER".STAT55_MAX_RAW_LHFD,
                               IN2 := "DB106_DATA_PARAMETER".STAT13_HAND_REFF_LHFD_FA,
                               Out15 => "DB140_ANALOG_OUTPUT"."STAT1_Speed LH FD Reff");
   END_IF;
END_REGION

REGION Network 20: UNSCALLING LSP(LOW SETPOINT) LHFD FAN | HMI | MIN RAW LH FD
   RUNG wire#powerrail
      "FC108_Unscalling_Custom"(IN0 := "DB106_DATA_PARAMETER".STAT20_LSP_LHFD_FAN, IN1 := 50.0, IN2 := 0.0, IN3 := "DB100_WORK_BIT".STAT57_ALWAYS_ON, IN4 := 0.0, IN5 := 27648.0, OUT_4 => "DB120_TEMP_DATA".STAT65)
      { S7_Templates := "[SrcType := Int, DestType := DInt]" } Convert(in := "DB120_TEMP_DATA".STAT65, out => "DB120_TEMP_DATA".STAT67)
      { S7_Templates := "[SrcType := DInt, DestType := Real]" } Convert(in := "DB120_TEMP_DATA".STAT67, out => "DB106_DATA_PARAMETER".STAT54_MIN_RAW_LHFD)
   END_RUNG
   // the same network as SCL:
   "FC108_Unscalling_Custom"(IN0 := "DB106_DATA_PARAMETER".STAT20_LSP_LHFD_FAN,
                           IN1 := 50.0,
                           IN2 := 0.0,
                           IN3 := "DB100_WORK_BIT".STAT57_ALWAYS_ON,
                           IN4 := 0.0,
                           IN5 := 27648.0,
                           OUT_4 => "DB120_TEMP_DATA".STAT65,
                           ENO => #_w1);
   IF #_w1 THEN
       "DB120_TEMP_DATA".STAT67 := INT_TO_DINT("DB120_TEMP_DATA".STAT65);
       "DB106_DATA_PARAMETER".STAT54_MIN_RAW_LHFD := DINT_TO_REAL("DB120_TEMP_DATA".STAT67);
   END_IF;
END_REGION

REGION Network 21: UNSCALLING HSP(HIGH SETPOINT) LHFD FAN | HMI | MAX RAW LH FD
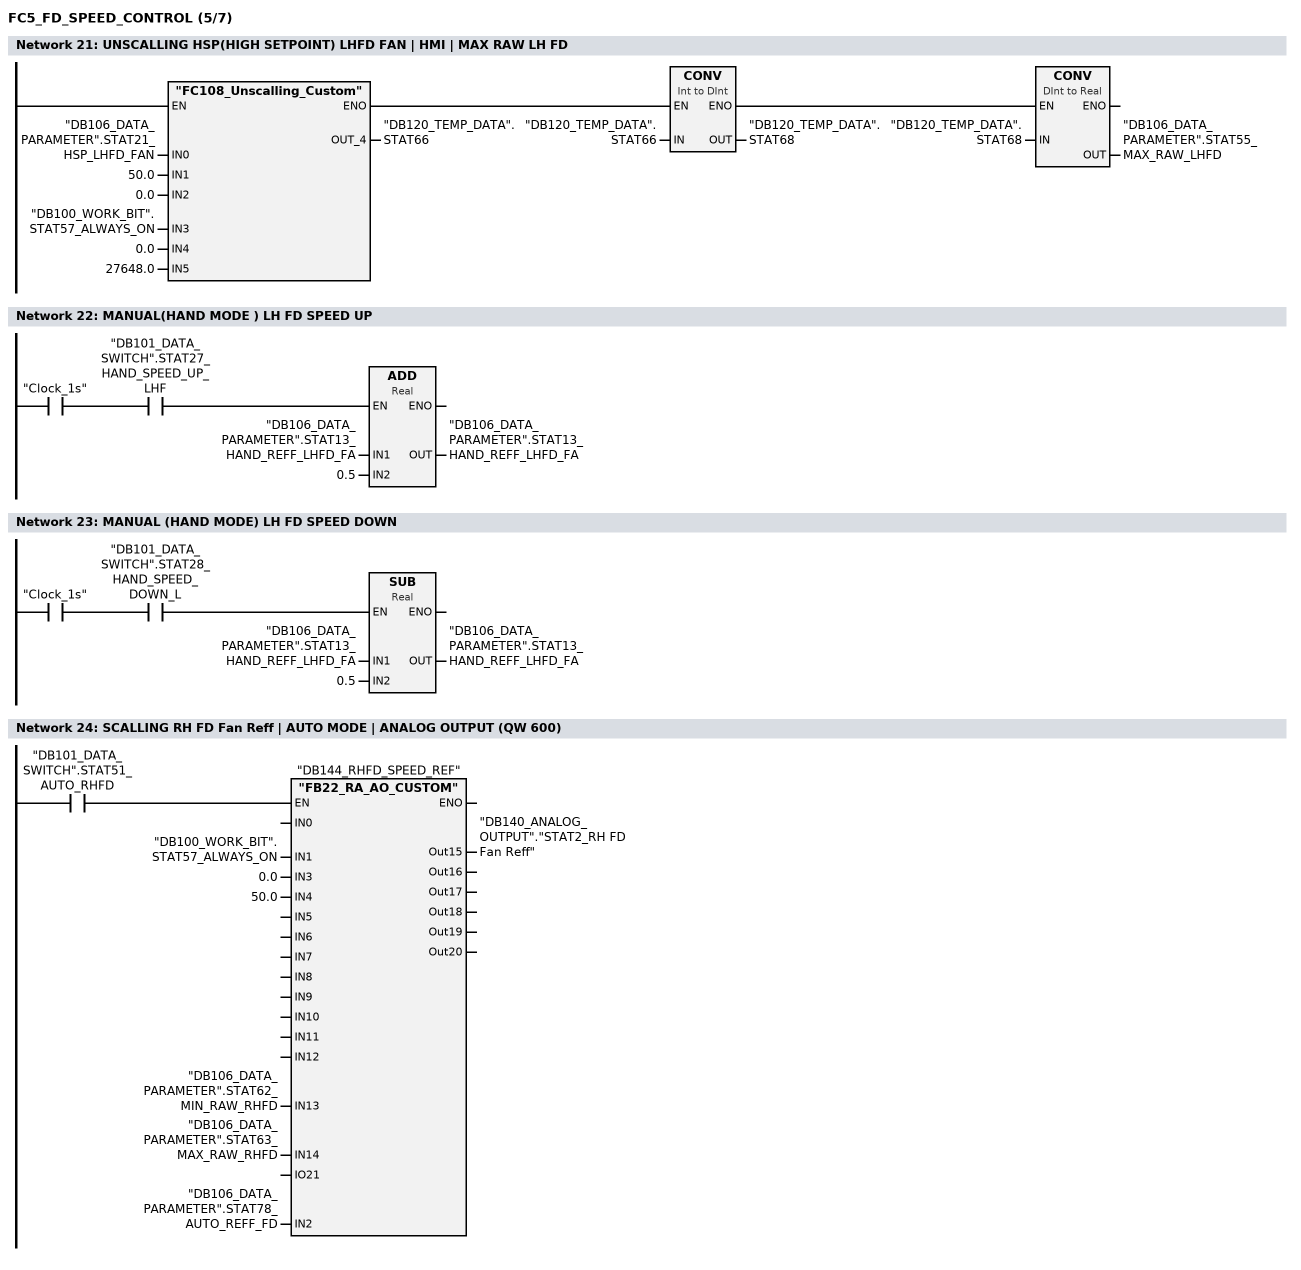
   RUNG wire#powerrail
      "FC108_Unscalling_Custom"(IN0 := "DB106_DATA_PARAMETER".STAT21_HSP_LHFD_FAN, IN1 := 50.0, IN2 := 0.0, IN3 := "DB100_WORK_BIT".STAT57_ALWAYS_ON, IN4 := 0.0, IN5 := 27648.0, OUT_4 => "DB120_TEMP_DATA".STAT66)
      { S7_Templates := "[SrcType := Int, DestType := DInt]" } Convert(in := "DB120_TEMP_DATA".STAT66, out => "DB120_TEMP_DATA".STAT68)
      { S7_Templates := "[SrcType := DInt, DestType := Real]" } Convert(in := "DB120_TEMP_DATA".STAT68, out => "DB106_DATA_PARAMETER".STAT55_MAX_RAW_LHFD)
   END_RUNG
   // the same network as SCL:
   "FC108_Unscalling_Custom"(IN0 := "DB106_DATA_PARAMETER".STAT21_HSP_LHFD_FAN,
                           IN1 := 50.0,
                           IN2 := 0.0,
                           IN3 := "DB100_WORK_BIT".STAT57_ALWAYS_ON,
                           IN4 := 0.0,
                           IN5 := 27648.0,
                           OUT_4 => "DB120_TEMP_DATA".STAT66,
                           ENO => #_w1);
   IF #_w1 THEN
       "DB120_TEMP_DATA".STAT68 := INT_TO_DINT("DB120_TEMP_DATA".STAT66);
       "DB106_DATA_PARAMETER".STAT55_MAX_RAW_LHFD := DINT_TO_REAL("DB120_TEMP_DATA".STAT68);
   END_IF;
END_REGION

REGION Network 22: MANUAL(HAND MODE ) LH FD SPEED UP
   RUNG wire#powerrail
      Contact( "Clock_1s" )
      Contact( "DB101_DATA_SWITCH".STAT27_HAND_SPEED_UP_LHF )
      { S7_Templates := "SrcType := Real" } Add(in1 := "DB106_DATA_PARAMETER".STAT13_HAND_REFF_LHFD_FA, in2 := 0.5, out => "DB106_DATA_PARAMETER".STAT13_HAND_REFF_LHFD_FA)
   END_RUNG
   // the same network as SCL:
   IF "Clock_1s" AND "DB101_DATA_SWITCH".STAT27_HAND_SPEED_UP_LHF THEN
       "DB106_DATA_PARAMETER".STAT13_HAND_REFF_LHFD_FA := "DB106_DATA_PARAMETER".STAT13_HAND_REFF_LHFD_FA + 0.5;
   END_IF;
END_REGION

REGION Network 23: MANUAL (HAND MODE) LH FD SPEED DOWN
   RUNG wire#powerrail
      Contact( "Clock_1s" )
      Contact( "DB101_DATA_SWITCH".STAT28_HAND_SPEED_DOWN_L )
      { S7_Templates := "SrcType := Real" } Sub(in1 := "DB106_DATA_PARAMETER".STAT13_HAND_REFF_LHFD_FA, in2 := 0.5, out => "DB106_DATA_PARAMETER".STAT13_HAND_REFF_LHFD_FA)
   END_RUNG
   // the same network as SCL:
   IF "Clock_1s" AND "DB101_DATA_SWITCH".STAT28_HAND_SPEED_DOWN_L THEN
       "DB106_DATA_PARAMETER".STAT13_HAND_REFF_LHFD_FA := "DB106_DATA_PARAMETER".STAT13_HAND_REFF_LHFD_FA - 0.5;
   END_IF;
END_REGION

REGION Network 24: SCALLING RH FD Fan Reff | AUTO MODE | ANALOG OUTPUT (QW 600)
   RUNG wire#powerrail
      Contact( "DB101_DATA_SWITCH".STAT51_AUTO_RHFD )
      "DB144_RHFD_SPEED_REF"(IN0 :=, IN1 := "DB100_WORK_BIT".STAT57_ALWAYS_ON, IN3 := 0.0, IN4 := 50.0, IN5 :=, IN6 :=, IN7 :=, IN8 :=, IN9 :=, IN10 :=, IN11 :=, IN12 :=, IN13 := "DB106_DATA_PARAMETER".STAT62_MIN_RAW_RHFD, IN14 := "DB106_DATA_PARAMETER".STAT63_MAX_RAW_RHFD, IO21 :=, IN2 := "DB106_DATA_PARAMETER".STAT78_AUTO_REFF_FD, Out15 => "DB140_ANALOG_OUTPUT"."STAT2_RH FD Fan Reff", Out16 =>, Out17 =>, Out18 =>, Out19 =>, Out20 =>)
   END_RUNG
   // the same network as SCL:
   IF "DB101_DATA_SWITCH".STAT51_AUTO_RHFD THEN
       "DB144_RHFD_SPEED_REF"(IN1 := "DB100_WORK_BIT".STAT57_ALWAYS_ON,   // "FB22_RA_AO_CUSTOM"
                              IN3 := 0.0,
                              IN4 := 50.0,
                              IN13 := "DB106_DATA_PARAMETER".STAT62_MIN_RAW_RHFD,
                              IN14 := "DB106_DATA_PARAMETER".STAT63_MAX_RAW_RHFD,
                              IN2 := "DB106_DATA_PARAMETER".STAT78_AUTO_REFF_FD,
                              Out15 => "DB140_ANALOG_OUTPUT"."STAT2_RH FD Fan Reff");
   END_IF;
END_REGION

REGION Network 25: SCALLING RH FD Fan Reff | MANUAL MODE | ANALOG OUTPUT (QW 600)
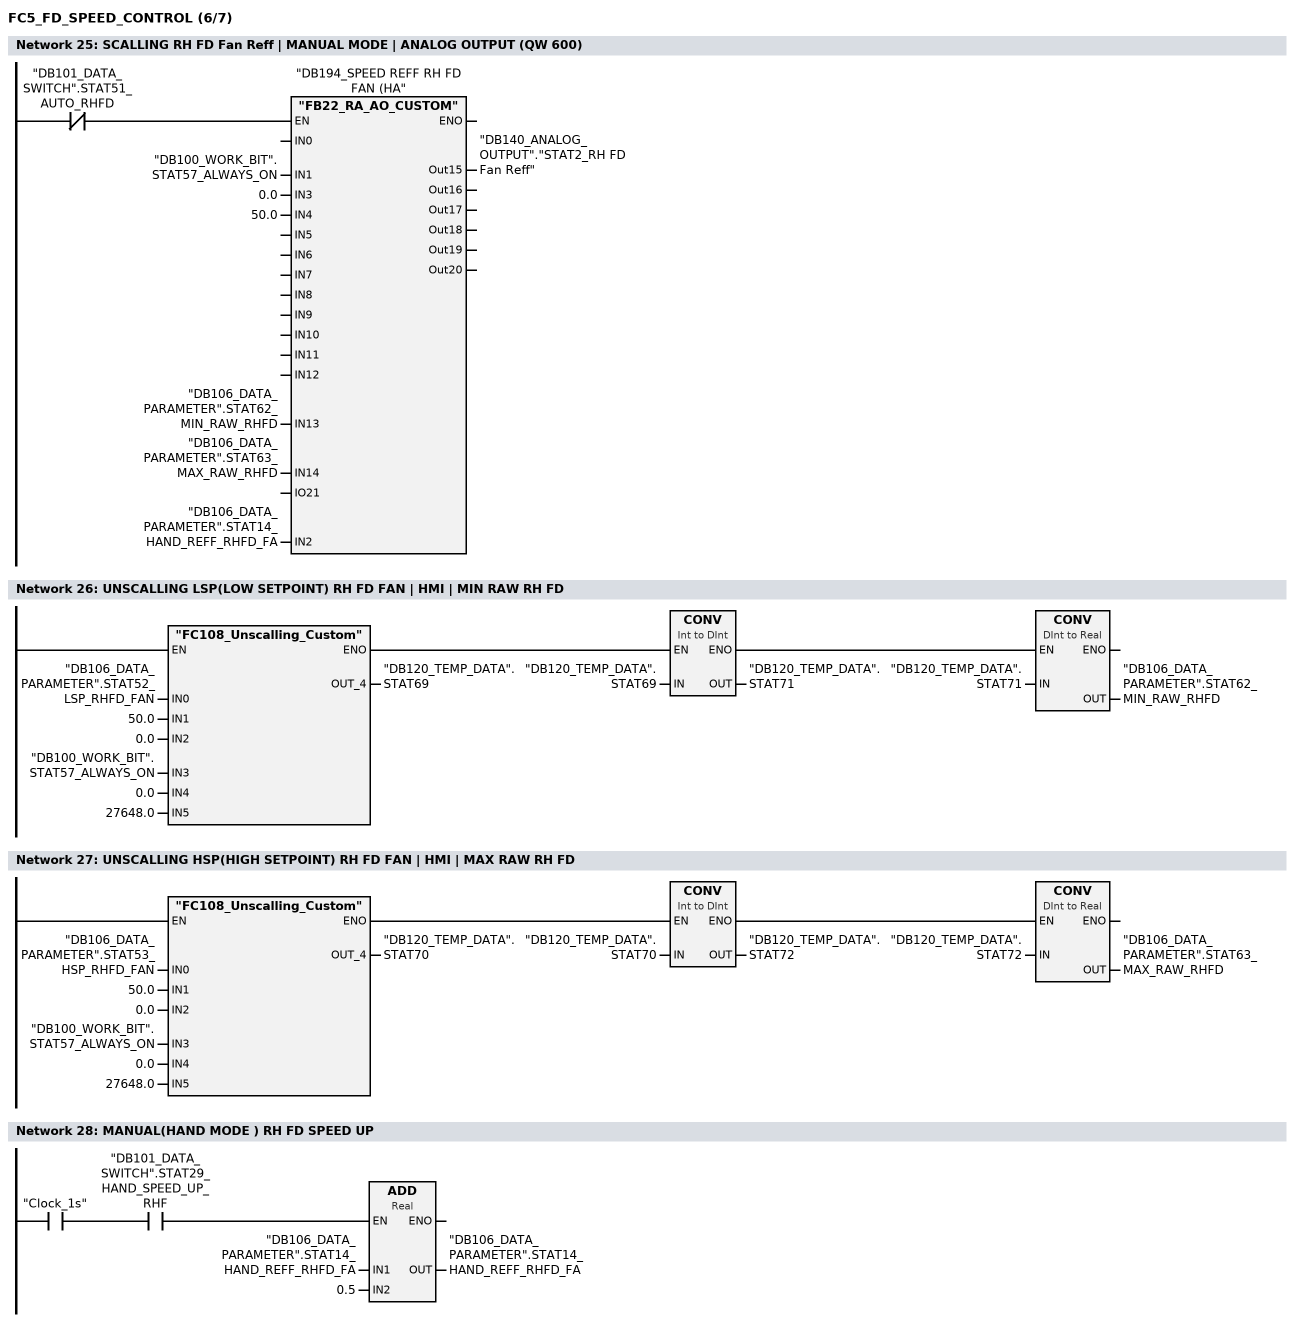
   RUNG wire#powerrail
      I_Contact( "DB101_DATA_SWITCH".STAT51_AUTO_RHFD )
      "DB194_SPEED REFF RH FD FAN (HA"(IN0 :=, IN1 := "DB100_WORK_BIT".STAT57_ALWAYS_ON, IN3 := 0.0, IN4 := 50.0, IN5 :=, IN6 :=, IN7 :=, IN8 :=, IN9 :=, IN10 :=, IN11 :=, IN12 :=, IN13 := "DB106_DATA_PARAMETER".STAT62_MIN_RAW_RHFD, IN14 := "DB106_DATA_PARAMETER".STAT63_MAX_RAW_RHFD, IO21 :=, IN2 := "DB106_DATA_PARAMETER".STAT14_HAND_REFF_RHFD_FA, Out15 => "DB140_ANALOG_OUTPUT"."STAT2_RH FD Fan Reff", Out16 =>, Out17 =>, Out18 =>, Out19 =>, Out20 =>)
   END_RUNG
   // the same network as SCL:
   IF NOT "DB101_DATA_SWITCH".STAT51_AUTO_RHFD THEN
       "DB194_SPEED REFF RH FD FAN (HA"(IN1 := "DB100_WORK_BIT".STAT57_ALWAYS_ON,   // "FB22_RA_AO_CUSTOM"
                               IN3 := 0.0,
                               IN4 := 50.0,
                               IN13 := "DB106_DATA_PARAMETER".STAT62_MIN_RAW_RHFD,
                               IN14 := "DB106_DATA_PARAMETER".STAT63_MAX_RAW_RHFD,
                               IN2 := "DB106_DATA_PARAMETER".STAT14_HAND_REFF_RHFD_FA,
                               Out15 => "DB140_ANALOG_OUTPUT"."STAT2_RH FD Fan Reff");
   END_IF;
END_REGION

REGION Network 26: UNSCALLING LSP(LOW SETPOINT) RH FD FAN | HMI | MIN RAW RH FD
   RUNG wire#powerrail
      "FC108_Unscalling_Custom"(IN0 := "DB106_DATA_PARAMETER".STAT52_LSP_RHFD_FAN, IN1 := 50.0, IN2 := 0.0, IN3 := "DB100_WORK_BIT".STAT57_ALWAYS_ON, IN4 := 0.0, IN5 := 27648.0, OUT_4 => "DB120_TEMP_DATA".STAT69)
      { S7_Templates := "[SrcType := Int, DestType := DInt]" } Convert(in := "DB120_TEMP_DATA".STAT69, out => "DB120_TEMP_DATA".STAT71)
      { S7_Templates := "[SrcType := DInt, DestType := Real]" } Convert(in := "DB120_TEMP_DATA".STAT71, out => "DB106_DATA_PARAMETER".STAT62_MIN_RAW_RHFD)
   END_RUNG
   // the same network as SCL:
   "FC108_Unscalling_Custom"(IN0 := "DB106_DATA_PARAMETER".STAT52_LSP_RHFD_FAN,
                           IN1 := 50.0,
                           IN2 := 0.0,
                           IN3 := "DB100_WORK_BIT".STAT57_ALWAYS_ON,
                           IN4 := 0.0,
                           IN5 := 27648.0,
                           OUT_4 => "DB120_TEMP_DATA".STAT69,
                           ENO => #_w1);
   IF #_w1 THEN
       "DB120_TEMP_DATA".STAT71 := INT_TO_DINT("DB120_TEMP_DATA".STAT69);
       "DB106_DATA_PARAMETER".STAT62_MIN_RAW_RHFD := DINT_TO_REAL("DB120_TEMP_DATA".STAT71);
   END_IF;
END_REGION

REGION Network 27: UNSCALLING HSP(HIGH SETPOINT) RH FD FAN | HMI | MAX RAW RH FD
   RUNG wire#powerrail
      "FC108_Unscalling_Custom"(IN0 := "DB106_DATA_PARAMETER".STAT53_HSP_RHFD_FAN, IN1 := 50.0, IN2 := 0.0, IN3 := "DB100_WORK_BIT".STAT57_ALWAYS_ON, IN4 := 0.0, IN5 := 27648.0, OUT_4 => "DB120_TEMP_DATA".STAT70)
      { S7_Templates := "[SrcType := Int, DestType := DInt]" } Convert(in := "DB120_TEMP_DATA".STAT70, out => "DB120_TEMP_DATA".STAT72)
      { S7_Templates := "[SrcType := DInt, DestType := Real]" } Convert(in := "DB120_TEMP_DATA".STAT72, out => "DB106_DATA_PARAMETER".STAT63_MAX_RAW_RHFD)
   END_RUNG
   // the same network as SCL:
   "FC108_Unscalling_Custom"(IN0 := "DB106_DATA_PARAMETER".STAT53_HSP_RHFD_FAN,
                           IN1 := 50.0,
                           IN2 := 0.0,
                           IN3 := "DB100_WORK_BIT".STAT57_ALWAYS_ON,
                           IN4 := 0.0,
                           IN5 := 27648.0,
                           OUT_4 => "DB120_TEMP_DATA".STAT70,
                           ENO => #_w1);
   IF #_w1 THEN
       "DB120_TEMP_DATA".STAT72 := INT_TO_DINT("DB120_TEMP_DATA".STAT70);
       "DB106_DATA_PARAMETER".STAT63_MAX_RAW_RHFD := DINT_TO_REAL("DB120_TEMP_DATA".STAT72);
   END_IF;
END_REGION

REGION Network 28: MANUAL(HAND MODE ) RH FD SPEED UP
   RUNG wire#powerrail
      Contact( "Clock_1s" )
      Contact( "DB101_DATA_SWITCH".STAT29_HAND_SPEED_UP_RHF )
      { S7_Templates := "SrcType := Real" } Add(in1 := "DB106_DATA_PARAMETER".STAT14_HAND_REFF_RHFD_FA, in2 := 0.5, out => "DB106_DATA_PARAMETER".STAT14_HAND_REFF_RHFD_FA)
   END_RUNG
   // the same network as SCL:
   IF "Clock_1s" AND "DB101_DATA_SWITCH".STAT29_HAND_SPEED_UP_RHF THEN
       "DB106_DATA_PARAMETER".STAT14_HAND_REFF_RHFD_FA := "DB106_DATA_PARAMETER".STAT14_HAND_REFF_RHFD_FA + 0.5;
   END_IF;
END_REGION

REGION Network 29: MANUAL(HAND MODE ) RH FD SPEED DOWN
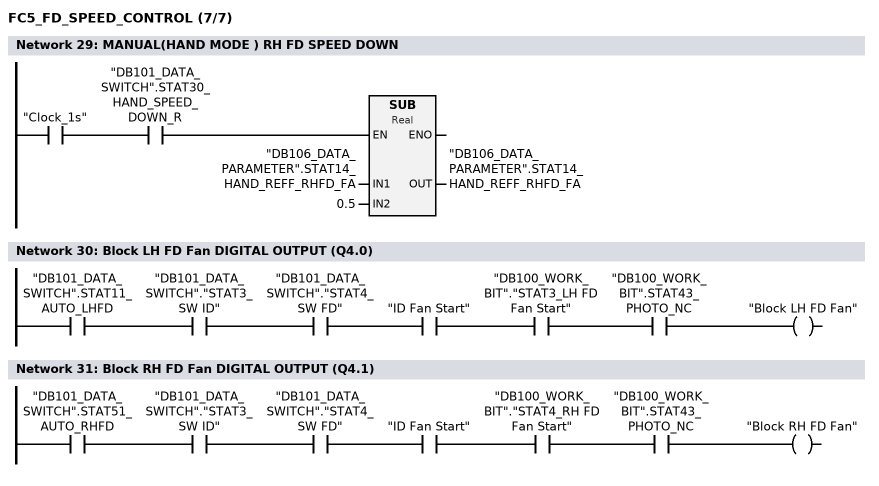
   RUNG wire#powerrail
      Contact( "Clock_1s" )
      Contact( "DB101_DATA_SWITCH".STAT30_HAND_SPEED_DOWN_R )
      { S7_Templates := "SrcType := Real" } Sub(in1 := "DB106_DATA_PARAMETER".STAT14_HAND_REFF_RHFD_FA, in2 := 0.5, out => "DB106_DATA_PARAMETER".STAT14_HAND_REFF_RHFD_FA)
   END_RUNG
   // the same network as SCL:
   IF "Clock_1s" AND "DB101_DATA_SWITCH".STAT30_HAND_SPEED_DOWN_R THEN
       "DB106_DATA_PARAMETER".STAT14_HAND_REFF_RHFD_FA := "DB106_DATA_PARAMETER".STAT14_HAND_REFF_RHFD_FA - 0.5;
   END_IF;
END_REGION

REGION Network 30: Block LH FD Fan DIGITAL OUTPUT (Q4.0)
   RUNG wire#powerrail
      Contact( "DB101_DATA_SWITCH".STAT11_AUTO_LHFD )
      Contact( "DB101_DATA_SWITCH"."STAT3_SW ID" )
      Contact( "DB101_DATA_SWITCH"."STAT4_SW FD" )
      Contact( "ID Fan Start" )
      Contact( "DB100_WORK_BIT"."STAT3_LH FD Fan Start" )
      Contact( "DB100_WORK_BIT".STAT43_PHOTO_NC )
      Coil( "Block LH FD Fan" )
   END_RUNG
   // the same network as SCL:
   "Block LH FD Fan" := "DB101_DATA_SWITCH".STAT11_AUTO_LHFD AND "DB101_DATA_SWITCH"."STAT3_SW ID" AND "DB101_DATA_SWITCH"."STAT4_SW FD" AND "ID Fan Start" AND "DB100_WORK_BIT"."STAT3_LH FD Fan Start" AND "DB100_WORK_BIT".STAT43_PHOTO_NC;
END_REGION

REGION Network 31: Block RH FD Fan DIGITAL OUTPUT (Q4.1)
   RUNG wire#powerrail
      Contact( "DB101_DATA_SWITCH".STAT51_AUTO_RHFD )
      Contact( "DB101_DATA_SWITCH"."STAT3_SW ID" )
      Contact( "DB101_DATA_SWITCH"."STAT4_SW FD" )
      Contact( "ID Fan Start" )
      Contact( "DB100_WORK_BIT"."STAT4_RH FD Fan Start" )
      Contact( "DB100_WORK_BIT".STAT43_PHOTO_NC )
      Coil( "Block RH FD Fan" )
   END_RUNG
   // the same network as SCL:
   "Block RH FD Fan" := "DB101_DATA_SWITCH".STAT51_AUTO_RHFD AND "DB101_DATA_SWITCH"."STAT3_SW ID" AND "DB101_DATA_SWITCH"."STAT4_SW FD" AND "ID Fan Start" AND "DB100_WORK_BIT"."STAT4_RH FD Fan Start" AND "DB100_WORK_BIT".STAT43_PHOTO_NC;
END_REGION
END_FUNCTION

FUNCTION "FC6_STOKER_SPEED_CONTROL" : Void   // FC6, LAD
TITLE = STOKER SPEED CONTROL
{ S7_Optimized_Access := 'TRUE' }
VERSION : 0.1
// INPUT PID  = IW 100
// 
// AO SPEED LH STOKER = QW 602
// AO SPEED RH STOKER = QW 604
// 
// DIGITAL OUPUT LH STOKER = Q0.5
// DIGITAL OUTPUT RH STOKER = Q0.6
   VAR_TEMP
      Out1 : DInt;
      Out2 : Real;
      Out3 : DInt;
      Out4 : Real;
      DIV1 : Real;
      DIV2 : Real;
   END_VAR
   VAR_TEMP   // added for the SCL form of the ladder/FBD networks
      _w1 : Bool;
   END_VAR
BEGIN

REGION Network 1: MOVE PARAMETER PID FROM HMI
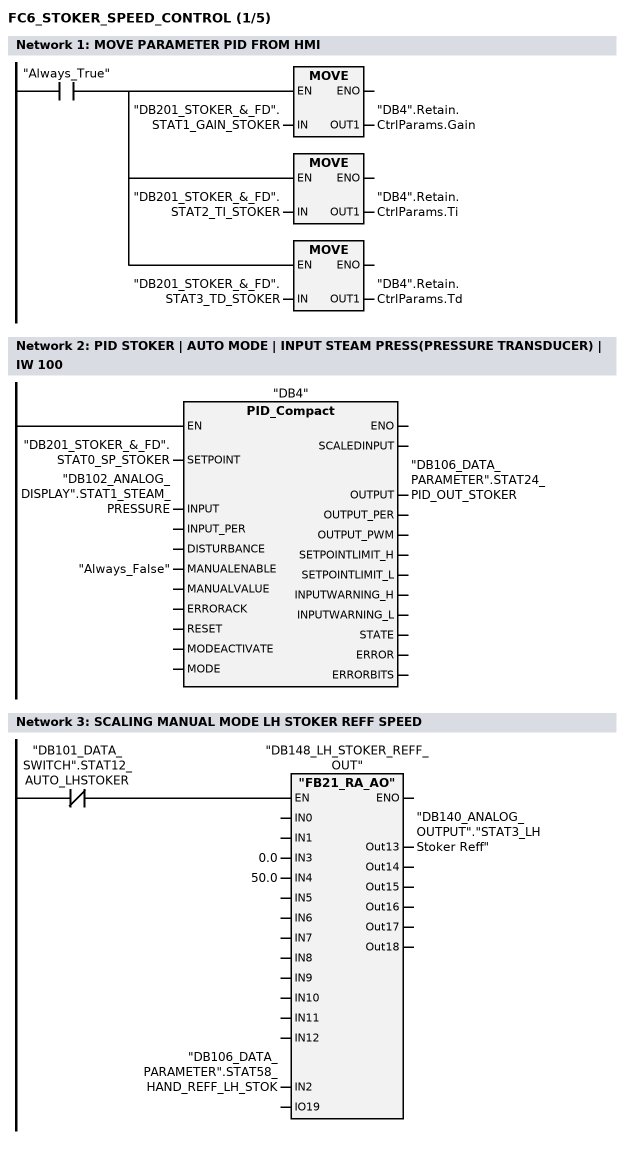
   RUNG wire#powerrail
      Contact( "Always_True" )
      wire#w1
      Move(in := "DB201_STOKER_&_FD".STAT1_GAIN_STOKER, out1 => "DB4".Retain.CtrlParams.Gain)
   END_RUNG
   RUNG wire#w1
      Move(in := "DB201_STOKER_&_FD".STAT2_TI_STOKER, out1 => "DB4".Retain.CtrlParams.Ti)
   END_RUNG
   RUNG wire#w1
      Move(in := "DB201_STOKER_&_FD".STAT3_TD_STOKER, out1 => "DB4".Retain.CtrlParams.Td)
   END_RUNG
   // the same network as SCL:
   IF "Always_True" THEN
       "DB4".Retain.CtrlParams.Gain := "DB201_STOKER_&_FD".STAT1_GAIN_STOKER;
       "DB4".Retain.CtrlParams.Ti := "DB201_STOKER_&_FD".STAT2_TI_STOKER;
       "DB4".Retain.CtrlParams.Td := "DB201_STOKER_&_FD".STAT3_TD_STOKER;
   END_IF;
END_REGION

REGION Network 2: PID STOKER | AUTO MODE | INPUT STEAM PRESS(PRESSURE TRANSDUCER) | IW 100
   "DB4"(Setpoint := "DB201_STOKER_&_FD".STAT0_SP_STOKER,   // PID_Compact
         Input := "DB102_ANALOG_DISPLAY".STAT1_STEAM_PRESSURE,
         ManualEnable := "Always_False",
         Output => "DB106_DATA_PARAMETER".STAT24_PID_OUT_STOKER);
END_REGION

REGION Network 3: SCALING MANUAL MODE LH STOKER REFF SPEED
   RUNG wire#powerrail
      I_Contact( "DB101_DATA_SWITCH".STAT12_AUTO_LHSTOKER )
      "DB148_LH_STOKER_REFF_OUT"(IN0 :=, IN1 :=, IN3 := 0.0, IN4 := 50.0, IN5 :=, IN6 :=, IN7 :=, IN8 :=, IN9 :=, IN10 :=, IN11 :=, IN12 :=, IN2 := "DB106_DATA_PARAMETER".STAT58_HAND_REFF_LH_STOK, IO19 :=, Out13 => "DB140_ANALOG_OUTPUT"."STAT3_LH Stoker Reff", Out14 =>, Out15 =>, Out16 =>, Out17 =>, Out18 =>)
   END_RUNG
   // the same network as SCL:
   IF NOT "DB101_DATA_SWITCH".STAT12_AUTO_LHSTOKER THEN
       "DB148_LH_STOKER_REFF_OUT"(IN3 := 0.0,   // "FB21_RA_AO"
                               IN4 := 50.0,
                               IN2 := "DB106_DATA_PARAMETER".STAT58_HAND_REFF_LH_STOK,
                               Out13 => "DB140_ANALOG_OUTPUT"."STAT3_LH Stoker Reff");
   END_IF;
END_REGION

REGION Network 4: SCALING AUTO MODE LH STOKER REFF SPEED
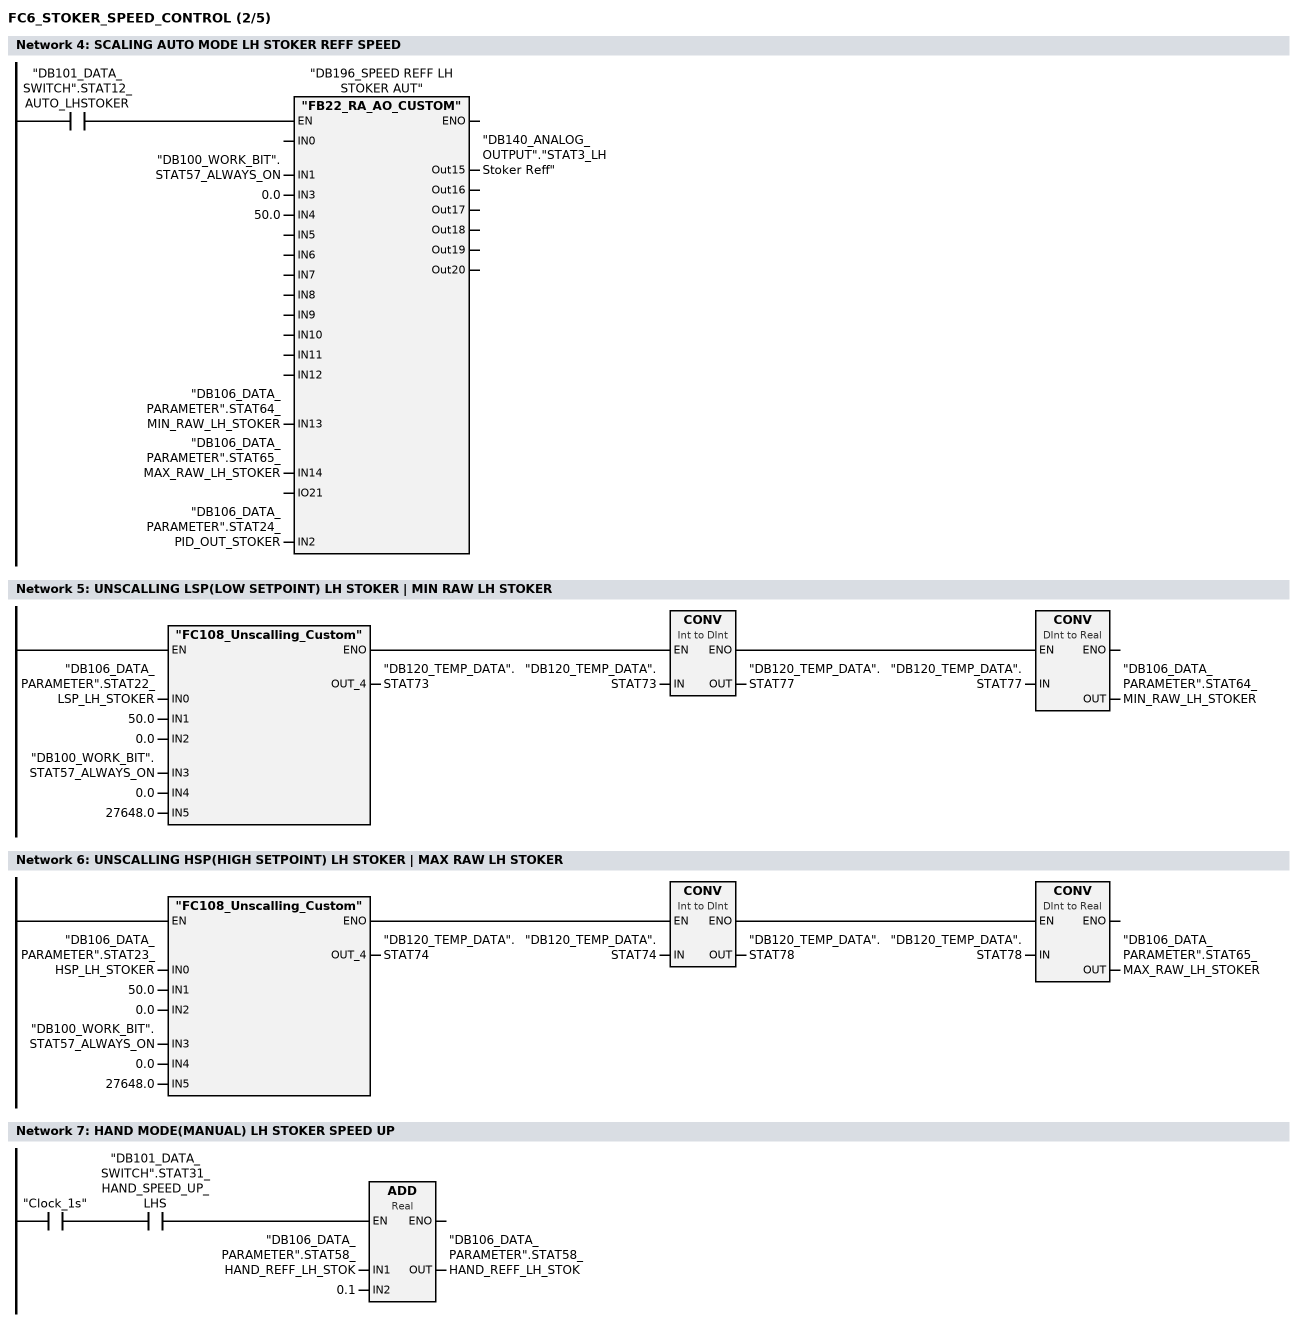
   RUNG wire#powerrail
      Contact( "DB101_DATA_SWITCH".STAT12_AUTO_LHSTOKER )
      "DB196_SPEED REFF LH STOKER AUT"(IN0 :=, IN1 := "DB100_WORK_BIT".STAT57_ALWAYS_ON, IN3 := 0.0, IN4 := 50.0, IN5 :=, IN6 :=, IN7 :=, IN8 :=, IN9 :=, IN10 :=, IN11 :=, IN12 :=, IN13 := "DB106_DATA_PARAMETER".STAT64_MIN_RAW_LH_STOKER, IN14 := "DB106_DATA_PARAMETER".STAT65_MAX_RAW_LH_STOKER, IO21 :=, IN2 := "DB106_DATA_PARAMETER".STAT24_PID_OUT_STOKER, Out15 => "DB140_ANALOG_OUTPUT"."STAT3_LH Stoker Reff", Out16 =>, Out17 =>, Out18 =>, Out19 =>, Out20 =>)
   END_RUNG
   // the same network as SCL:
   IF "DB101_DATA_SWITCH".STAT12_AUTO_LHSTOKER THEN
       "DB196_SPEED REFF LH STOKER AUT"(IN1 := "DB100_WORK_BIT".STAT57_ALWAYS_ON,   // "FB22_RA_AO_CUSTOM"
                               IN3 := 0.0,
                               IN4 := 50.0,
                               IN13 := "DB106_DATA_PARAMETER".STAT64_MIN_RAW_LH_STOKER,
                               IN14 := "DB106_DATA_PARAMETER".STAT65_MAX_RAW_LH_STOKER,
                               IN2 := "DB106_DATA_PARAMETER".STAT24_PID_OUT_STOKER,
                               Out15 => "DB140_ANALOG_OUTPUT"."STAT3_LH Stoker Reff");
   END_IF;
END_REGION

REGION Network 5: UNSCALLING LSP(LOW SETPOINT) LH STOKER | MIN RAW LH STOKER
   RUNG wire#powerrail
      "FC108_Unscalling_Custom"(IN0 := "DB106_DATA_PARAMETER".STAT22_LSP_LH_STOKER, IN1 := 50.0, IN2 := 0.0, IN3 := "DB100_WORK_BIT".STAT57_ALWAYS_ON, IN4 := 0.0, IN5 := 27648.0, OUT_4 => "DB120_TEMP_DATA".STAT73)
      { S7_Templates := "[SrcType := Int, DestType := DInt]" } Convert(in := "DB120_TEMP_DATA".STAT73, out => "DB120_TEMP_DATA".STAT77)
      { S7_Templates := "[SrcType := DInt, DestType := Real]" } Convert(in := "DB120_TEMP_DATA".STAT77, out => "DB106_DATA_PARAMETER".STAT64_MIN_RAW_LH_STOKER)
   END_RUNG
   // the same network as SCL:
   "FC108_Unscalling_Custom"(IN0 := "DB106_DATA_PARAMETER".STAT22_LSP_LH_STOKER,
                           IN1 := 50.0,
                           IN2 := 0.0,
                           IN3 := "DB100_WORK_BIT".STAT57_ALWAYS_ON,
                           IN4 := 0.0,
                           IN5 := 27648.0,
                           OUT_4 => "DB120_TEMP_DATA".STAT73,
                           ENO => #_w1);
   IF #_w1 THEN
       "DB120_TEMP_DATA".STAT77 := INT_TO_DINT("DB120_TEMP_DATA".STAT73);
       "DB106_DATA_PARAMETER".STAT64_MIN_RAW_LH_STOKER := DINT_TO_REAL("DB120_TEMP_DATA".STAT77);
   END_IF;
END_REGION

REGION Network 6: UNSCALLING HSP(HIGH SETPOINT) LH STOKER | MAX RAW LH STOKER
   RUNG wire#powerrail
      "FC108_Unscalling_Custom"(IN0 := "DB106_DATA_PARAMETER".STAT23_HSP_LH_STOKER, IN1 := 50.0, IN2 := 0.0, IN3 := "DB100_WORK_BIT".STAT57_ALWAYS_ON, IN4 := 0.0, IN5 := 27648.0, OUT_4 => "DB120_TEMP_DATA".STAT74)
      { S7_Templates := "[SrcType := Int, DestType := DInt]" } Convert(in := "DB120_TEMP_DATA".STAT74, out => "DB120_TEMP_DATA".STAT78)
      { S7_Templates := "[SrcType := DInt, DestType := Real]" } Convert(in := "DB120_TEMP_DATA".STAT78, out => "DB106_DATA_PARAMETER".STAT65_MAX_RAW_LH_STOKER)
   END_RUNG
   // the same network as SCL:
   "FC108_Unscalling_Custom"(IN0 := "DB106_DATA_PARAMETER".STAT23_HSP_LH_STOKER,
                           IN1 := 50.0,
                           IN2 := 0.0,
                           IN3 := "DB100_WORK_BIT".STAT57_ALWAYS_ON,
                           IN4 := 0.0,
                           IN5 := 27648.0,
                           OUT_4 => "DB120_TEMP_DATA".STAT74,
                           ENO => #_w1);
   IF #_w1 THEN
       "DB120_TEMP_DATA".STAT78 := INT_TO_DINT("DB120_TEMP_DATA".STAT74);
       "DB106_DATA_PARAMETER".STAT65_MAX_RAW_LH_STOKER := DINT_TO_REAL("DB120_TEMP_DATA".STAT78);
   END_IF;
END_REGION

REGION Network 7: HAND MODE(MANUAL) LH STOKER SPEED UP
   RUNG wire#powerrail
      Contact( "Clock_1s" )
      Contact( "DB101_DATA_SWITCH".STAT31_HAND_SPEED_UP_LHS )
      { S7_Templates := "SrcType := Real" } Add(in1 := "DB106_DATA_PARAMETER".STAT58_HAND_REFF_LH_STOK, in2 := 0.1, out => "DB106_DATA_PARAMETER".STAT58_HAND_REFF_LH_STOK)
   END_RUNG
   // the same network as SCL:
   IF "Clock_1s" AND "DB101_DATA_SWITCH".STAT31_HAND_SPEED_UP_LHS THEN
       "DB106_DATA_PARAMETER".STAT58_HAND_REFF_LH_STOK := "DB106_DATA_PARAMETER".STAT58_HAND_REFF_LH_STOK + 0.1;
   END_IF;
END_REGION

REGION Network 8: HAND MODE(MANUAL) LH STOKER SPEED DOWN
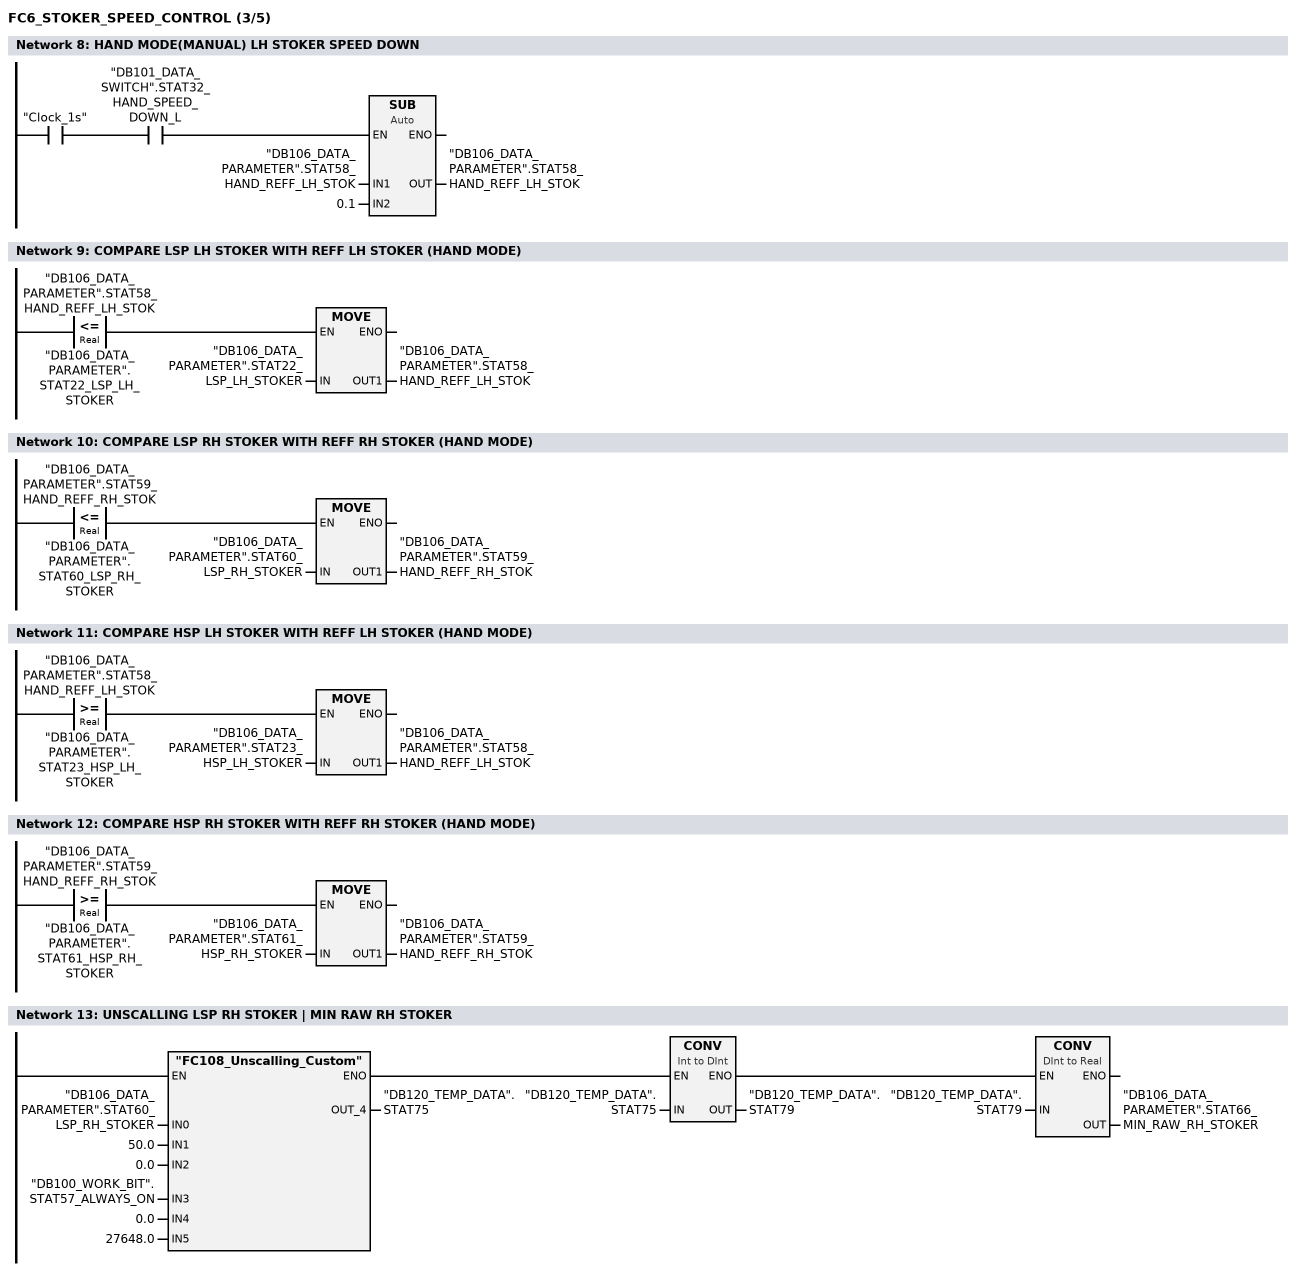
   RUNG wire#powerrail
      Contact( "Clock_1s" )
      Contact( "DB101_DATA_SWITCH".STAT32_HAND_SPEED_DOWN_L )
      Sub(in1 := "DB106_DATA_PARAMETER".STAT58_HAND_REFF_LH_STOK, in2 := 0.1, out => "DB106_DATA_PARAMETER".STAT58_HAND_REFF_LH_STOK)
   END_RUNG
   // the same network as SCL:
   IF "Clock_1s" AND "DB101_DATA_SWITCH".STAT32_HAND_SPEED_DOWN_L THEN
       "DB106_DATA_PARAMETER".STAT58_HAND_REFF_LH_STOK := "DB106_DATA_PARAMETER".STAT58_HAND_REFF_LH_STOK - 0.1;
   END_IF;
END_REGION

REGION Network 9: COMPARE LSP LH STOKER WITH REFF LH STOKER (HAND MODE)
   RUNG wire#powerrail
      { S7_Templates := "SrcType := Real" } LE_Contact(in1 := "DB106_DATA_PARAMETER".STAT58_HAND_REFF_LH_STOK, in2 := "DB106_DATA_PARAMETER".STAT22_LSP_LH_STOKER)
      Move(in := "DB106_DATA_PARAMETER".STAT22_LSP_LH_STOKER, out1 => "DB106_DATA_PARAMETER".STAT58_HAND_REFF_LH_STOK)
   END_RUNG
   // the same network as SCL:
   IF "DB106_DATA_PARAMETER".STAT58_HAND_REFF_LH_STOK <= "DB106_DATA_PARAMETER".STAT22_LSP_LH_STOKER THEN
       "DB106_DATA_PARAMETER".STAT58_HAND_REFF_LH_STOK := "DB106_DATA_PARAMETER".STAT22_LSP_LH_STOKER;
   END_IF;
END_REGION

REGION Network 10: COMPARE LSP RH STOKER WITH REFF RH STOKER (HAND MODE)
   RUNG wire#powerrail
      { S7_Templates := "SrcType := Real" } LE_Contact(in1 := "DB106_DATA_PARAMETER".STAT59_HAND_REFF_RH_STOK, in2 := "DB106_DATA_PARAMETER".STAT60_LSP_RH_STOKER)
      Move(in := "DB106_DATA_PARAMETER".STAT60_LSP_RH_STOKER, out1 => "DB106_DATA_PARAMETER".STAT59_HAND_REFF_RH_STOK)
   END_RUNG
   // the same network as SCL:
   IF "DB106_DATA_PARAMETER".STAT59_HAND_REFF_RH_STOK <= "DB106_DATA_PARAMETER".STAT60_LSP_RH_STOKER THEN
       "DB106_DATA_PARAMETER".STAT59_HAND_REFF_RH_STOK := "DB106_DATA_PARAMETER".STAT60_LSP_RH_STOKER;
   END_IF;
END_REGION

REGION Network 11: COMPARE HSP LH STOKER WITH REFF LH STOKER (HAND MODE)
   RUNG wire#powerrail
      { S7_Templates := "SrcType := Real" } GE_Contact(in1 := "DB106_DATA_PARAMETER".STAT58_HAND_REFF_LH_STOK, in2 := "DB106_DATA_PARAMETER".STAT23_HSP_LH_STOKER)
      Move(in := "DB106_DATA_PARAMETER".STAT23_HSP_LH_STOKER, out1 => "DB106_DATA_PARAMETER".STAT58_HAND_REFF_LH_STOK)
   END_RUNG
   // the same network as SCL:
   IF "DB106_DATA_PARAMETER".STAT58_HAND_REFF_LH_STOK >= "DB106_DATA_PARAMETER".STAT23_HSP_LH_STOKER THEN
       "DB106_DATA_PARAMETER".STAT58_HAND_REFF_LH_STOK := "DB106_DATA_PARAMETER".STAT23_HSP_LH_STOKER;
   END_IF;
END_REGION

REGION Network 12: COMPARE HSP RH STOKER WITH REFF RH STOKER (HAND MODE)
   RUNG wire#powerrail
      { S7_Templates := "SrcType := Real" } GE_Contact(in1 := "DB106_DATA_PARAMETER".STAT59_HAND_REFF_RH_STOK, in2 := "DB106_DATA_PARAMETER".STAT61_HSP_RH_STOKER)
      Move(in := "DB106_DATA_PARAMETER".STAT61_HSP_RH_STOKER, out1 => "DB106_DATA_PARAMETER".STAT59_HAND_REFF_RH_STOK)
   END_RUNG
   // the same network as SCL:
   IF "DB106_DATA_PARAMETER".STAT59_HAND_REFF_RH_STOK >= "DB106_DATA_PARAMETER".STAT61_HSP_RH_STOKER THEN
       "DB106_DATA_PARAMETER".STAT59_HAND_REFF_RH_STOK := "DB106_DATA_PARAMETER".STAT61_HSP_RH_STOKER;
   END_IF;
END_REGION

REGION Network 13: UNSCALLING LSP RH STOKER | MIN RAW RH STOKER
   RUNG wire#powerrail
      "FC108_Unscalling_Custom"(IN0 := "DB106_DATA_PARAMETER".STAT60_LSP_RH_STOKER, IN1 := 50.0, IN2 := 0.0, IN3 := "DB100_WORK_BIT".STAT57_ALWAYS_ON, IN4 := 0.0, IN5 := 27648.0, OUT_4 => "DB120_TEMP_DATA".STAT75)
      { S7_Templates := "[SrcType := Int, DestType := DInt]" } Convert(in := "DB120_TEMP_DATA".STAT75, out => "DB120_TEMP_DATA".STAT79)
      { S7_Templates := "[SrcType := DInt, DestType := Real]" } Convert(in := "DB120_TEMP_DATA".STAT79, out => "DB106_DATA_PARAMETER".STAT66_MIN_RAW_RH_STOKER)
   END_RUNG
   // the same network as SCL:
   "FC108_Unscalling_Custom"(IN0 := "DB106_DATA_PARAMETER".STAT60_LSP_RH_STOKER,
                           IN1 := 50.0,
                           IN2 := 0.0,
                           IN3 := "DB100_WORK_BIT".STAT57_ALWAYS_ON,
                           IN4 := 0.0,
                           IN5 := 27648.0,
                           OUT_4 => "DB120_TEMP_DATA".STAT75,
                           ENO => #_w1);
   IF #_w1 THEN
       "DB120_TEMP_DATA".STAT79 := INT_TO_DINT("DB120_TEMP_DATA".STAT75);
       "DB106_DATA_PARAMETER".STAT66_MIN_RAW_RH_STOKER := DINT_TO_REAL("DB120_TEMP_DATA".STAT79);
   END_IF;
END_REGION

REGION Network 14: UNSCALLING HSP RH STOKER | MAX RAW RH STOKER
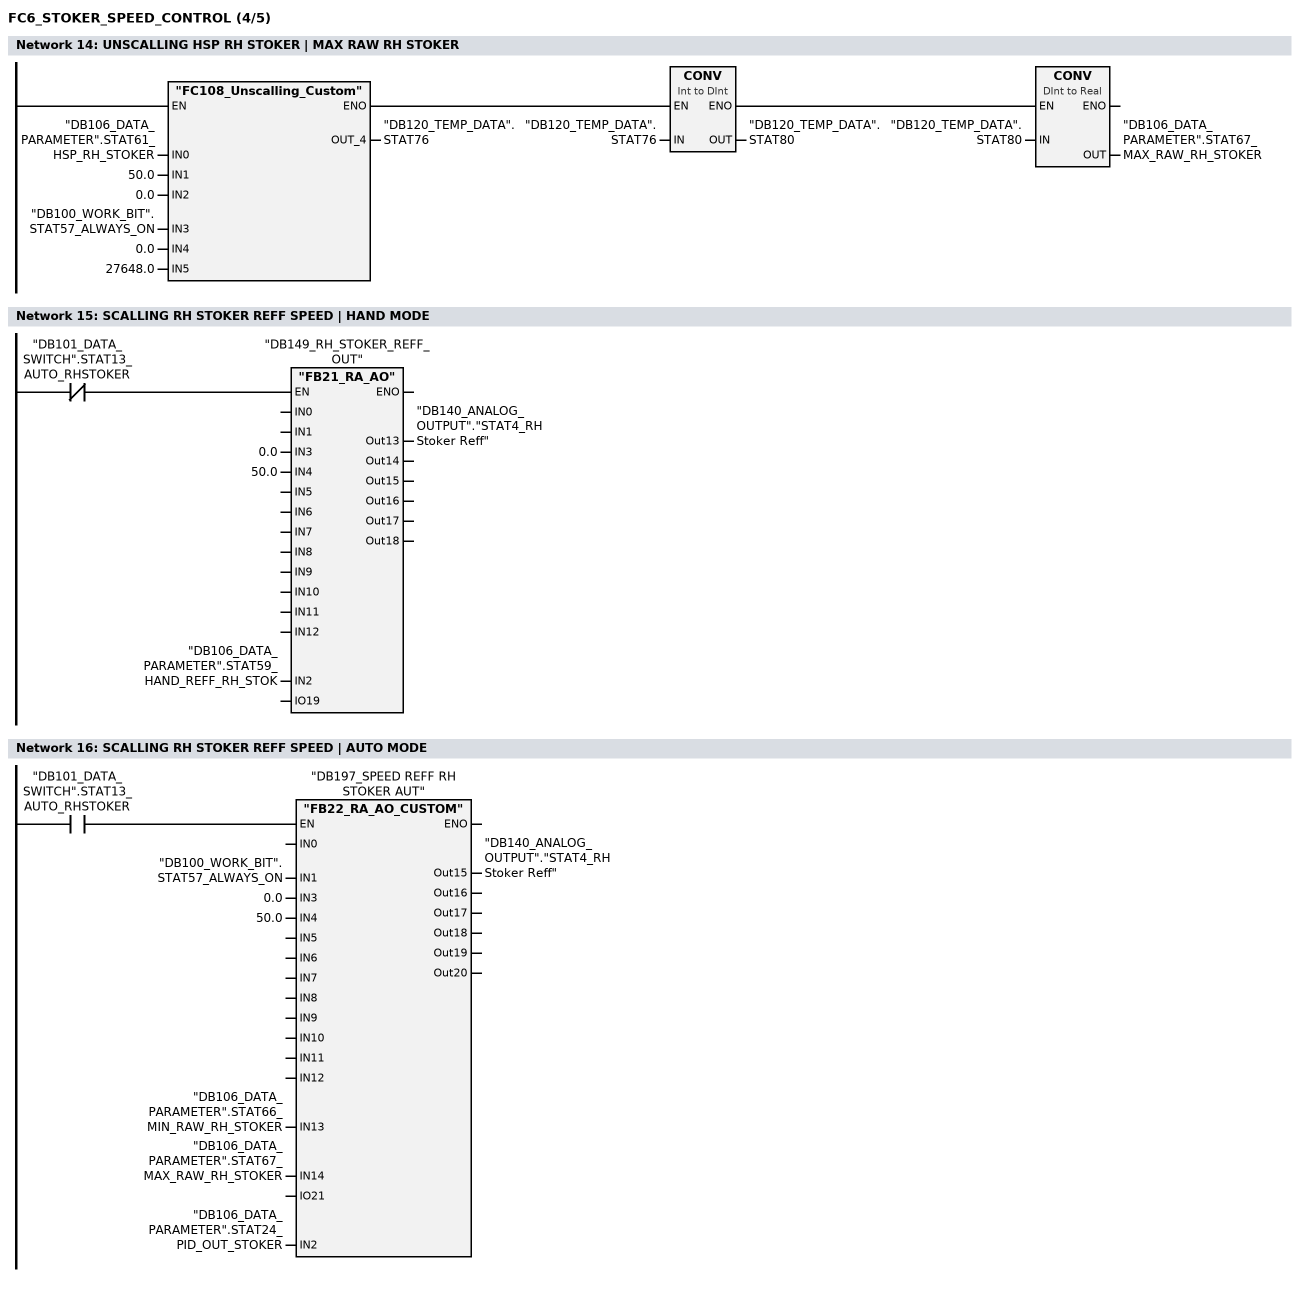
   RUNG wire#powerrail
      "FC108_Unscalling_Custom"(IN0 := "DB106_DATA_PARAMETER".STAT61_HSP_RH_STOKER, IN1 := 50.0, IN2 := 0.0, IN3 := "DB100_WORK_BIT".STAT57_ALWAYS_ON, IN4 := 0.0, IN5 := 27648.0, OUT_4 => "DB120_TEMP_DATA".STAT76)
      { S7_Templates := "[SrcType := Int, DestType := DInt]" } Convert(in := "DB120_TEMP_DATA".STAT76, out => "DB120_TEMP_DATA".STAT80)
      { S7_Templates := "[SrcType := DInt, DestType := Real]" } Convert(in := "DB120_TEMP_DATA".STAT80, out => "DB106_DATA_PARAMETER".STAT67_MAX_RAW_RH_STOKER)
   END_RUNG
   // the same network as SCL:
   "FC108_Unscalling_Custom"(IN0 := "DB106_DATA_PARAMETER".STAT61_HSP_RH_STOKER,
                           IN1 := 50.0,
                           IN2 := 0.0,
                           IN3 := "DB100_WORK_BIT".STAT57_ALWAYS_ON,
                           IN4 := 0.0,
                           IN5 := 27648.0,
                           OUT_4 => "DB120_TEMP_DATA".STAT76,
                           ENO => #_w1);
   IF #_w1 THEN
       "DB120_TEMP_DATA".STAT80 := INT_TO_DINT("DB120_TEMP_DATA".STAT76);
       "DB106_DATA_PARAMETER".STAT67_MAX_RAW_RH_STOKER := DINT_TO_REAL("DB120_TEMP_DATA".STAT80);
   END_IF;
END_REGION

REGION Network 15: SCALLING RH STOKER REFF SPEED | HAND MODE
   RUNG wire#powerrail
      I_Contact( "DB101_DATA_SWITCH".STAT13_AUTO_RHSTOKER )
      "DB149_RH_STOKER_REFF_OUT"(IN0 :=, IN1 :=, IN3 := 0.0, IN4 := 50.0, IN5 :=, IN6 :=, IN7 :=, IN8 :=, IN9 :=, IN10 :=, IN11 :=, IN12 :=, IN2 := "DB106_DATA_PARAMETER".STAT59_HAND_REFF_RH_STOK, IO19 :=, Out13 => "DB140_ANALOG_OUTPUT"."STAT4_RH Stoker Reff", Out14 =>, Out15 =>, Out16 =>, Out17 =>, Out18 =>)
   END_RUNG
   // the same network as SCL:
   IF NOT "DB101_DATA_SWITCH".STAT13_AUTO_RHSTOKER THEN
       "DB149_RH_STOKER_REFF_OUT"(IN3 := 0.0,   // "FB21_RA_AO"
                               IN4 := 50.0,
                               IN2 := "DB106_DATA_PARAMETER".STAT59_HAND_REFF_RH_STOK,
                               Out13 => "DB140_ANALOG_OUTPUT"."STAT4_RH Stoker Reff");
   END_IF;
END_REGION

REGION Network 16: SCALLING RH STOKER REFF SPEED | AUTO MODE
   RUNG wire#powerrail
      Contact( "DB101_DATA_SWITCH".STAT13_AUTO_RHSTOKER )
      "DB197_SPEED REFF RH STOKER AUT"(IN0 :=, IN1 := "DB100_WORK_BIT".STAT57_ALWAYS_ON, IN3 := 0.0, IN4 := 50.0, IN5 :=, IN6 :=, IN7 :=, IN8 :=, IN9 :=, IN10 :=, IN11 :=, IN12 :=, IN13 := "DB106_DATA_PARAMETER".STAT66_MIN_RAW_RH_STOKER, IN14 := "DB106_DATA_PARAMETER".STAT67_MAX_RAW_RH_STOKER, IO21 :=, IN2 := "DB106_DATA_PARAMETER".STAT24_PID_OUT_STOKER, Out15 => "DB140_ANALOG_OUTPUT"."STAT4_RH Stoker Reff", Out16 =>, Out17 =>, Out18 =>, Out19 =>, Out20 =>)
   END_RUNG
   // the same network as SCL:
   IF "DB101_DATA_SWITCH".STAT13_AUTO_RHSTOKER THEN
       "DB197_SPEED REFF RH STOKER AUT"(IN1 := "DB100_WORK_BIT".STAT57_ALWAYS_ON,   // "FB22_RA_AO_CUSTOM"
                               IN3 := 0.0,
                               IN4 := 50.0,
                               IN13 := "DB106_DATA_PARAMETER".STAT66_MIN_RAW_RH_STOKER,
                               IN14 := "DB106_DATA_PARAMETER".STAT67_MAX_RAW_RH_STOKER,
                               IN2 := "DB106_DATA_PARAMETER".STAT24_PID_OUT_STOKER,
                               Out15 => "DB140_ANALOG_OUTPUT"."STAT4_RH Stoker Reff");
   END_IF;
END_REGION

REGION Network 17: HAND MODE | REFF SPEED RH STOKER | SPEED UP
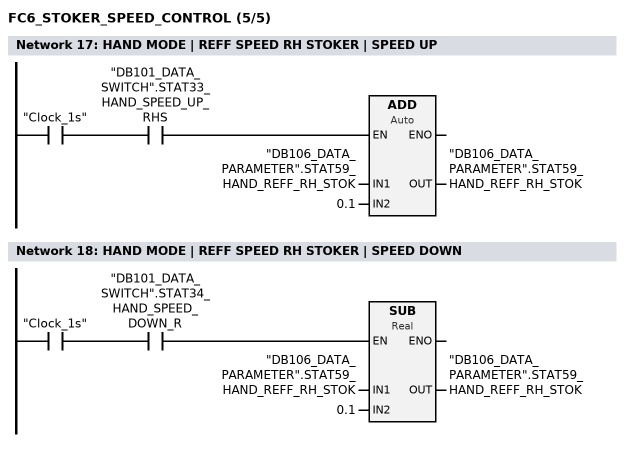
   RUNG wire#powerrail
      Contact( "Clock_1s" )
      Contact( "DB101_DATA_SWITCH".STAT33_HAND_SPEED_UP_RHS )
      Add(in1 := "DB106_DATA_PARAMETER".STAT59_HAND_REFF_RH_STOK, in2 := 0.1, out => "DB106_DATA_PARAMETER".STAT59_HAND_REFF_RH_STOK)
   END_RUNG
   // the same network as SCL:
   IF "Clock_1s" AND "DB101_DATA_SWITCH".STAT33_HAND_SPEED_UP_RHS THEN
       "DB106_DATA_PARAMETER".STAT59_HAND_REFF_RH_STOK := "DB106_DATA_PARAMETER".STAT59_HAND_REFF_RH_STOK + 0.1;
   END_IF;
END_REGION

REGION Network 18: HAND MODE | REFF SPEED RH STOKER | SPEED DOWN
   RUNG wire#powerrail
      Contact( "Clock_1s" )
      Contact( "DB101_DATA_SWITCH".STAT34_HAND_SPEED_DOWN_R )
      { S7_Templates := "SrcType := Real" } Sub(in1 := "DB106_DATA_PARAMETER".STAT59_HAND_REFF_RH_STOK, in2 := 0.1, out => "DB106_DATA_PARAMETER".STAT59_HAND_REFF_RH_STOK)
   END_RUNG
   // the same network as SCL:
   IF "Clock_1s" AND "DB101_DATA_SWITCH".STAT34_HAND_SPEED_DOWN_R THEN
       "DB106_DATA_PARAMETER".STAT59_HAND_REFF_RH_STOK := "DB106_DATA_PARAMETER".STAT59_HAND_REFF_RH_STOK - 0.1;
   END_IF;
END_REGION
END_FUNCTION

FUNCTION "FC7_WATER_FLOW_METER" : Void   // FC7, LAD
TITLE = WATER FLOW METER
{ S7_Optimized_Access := 'TRUE' }
VERSION : 0.1
// IW 104 = WATER FLOWRATE
// 
// I0.2 = WATER PULSER
   VAR_TEMP   // added for the SCL form of the ladder/FBD networks
      _w1 : Bool;
   END_VAR
BEGIN

REGION Network 1: SCALLING WATER FLOW RATE IW 104
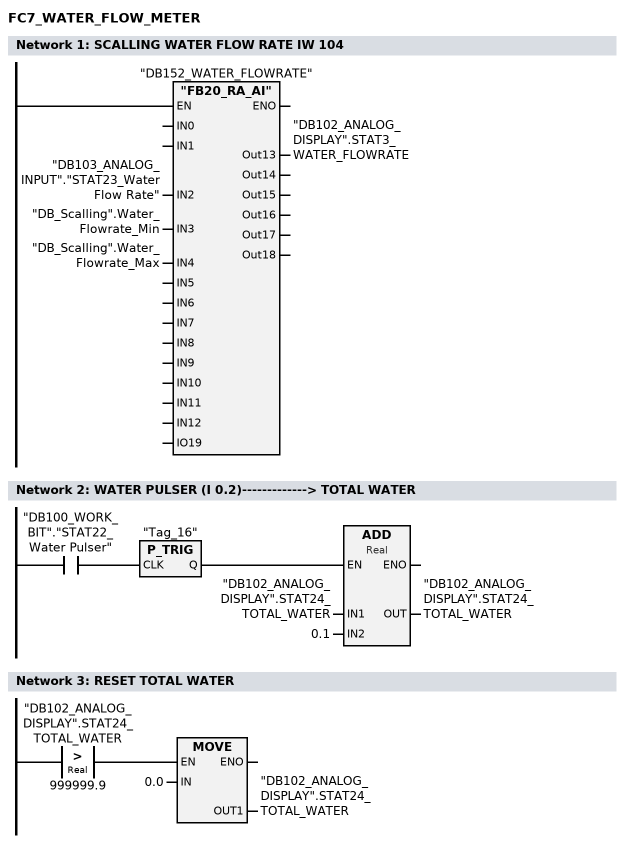
   RUNG wire#powerrail
      "DB152_WATER_FLOWRATE"(IN0 :=, IN1 :=, IN2 := "DB103_ANALOG_INPUT"."STAT23_Water Flow Rate", IN3 := "DB_Scalling".Water_Flowrate_Min, IN4 := "DB_Scalling".Water_Flowrate_Max, IN5 :=, IN6 :=, IN7 :=, IN8 :=, IN9 :=, IN10 :=, IN11 :=, IN12 :=, IO19 :=, Out13 => "DB102_ANALOG_DISPLAY".STAT3_WATER_FLOWRATE, Out14 =>, Out15 =>, Out16 =>, Out17 =>, Out18 =>)
   END_RUNG
   // the same network as SCL:
   "DB152_WATER_FLOWRATE"(IN2 := "DB103_ANALOG_INPUT"."STAT23_Water Flow Rate",   // "FB20_RA_AI"
                          IN3 := "DB_Scalling".Water_Flowrate_Min,
                          IN4 := "DB_Scalling".Water_Flowrate_Max,
                          Out13 => "DB102_ANALOG_DISPLAY".STAT3_WATER_FLOWRATE);
END_REGION

REGION Network 2: WATER PULSER (I 0.2)-------------> TOTAL WATER
   RUNG wire#powerrail
      Contact( "DB100_WORK_BIT"."STAT22_Water Pulser" )
      P_Trig( "Tag_16" )
      { S7_Templates := "SrcType := Real" } Add(in1 := "DB102_ANALOG_DISPLAY".STAT24_TOTAL_WATER, in2 := 0.1, out => "DB102_ANALOG_DISPLAY".STAT24_TOTAL_WATER)
   END_RUNG
   // the same network as SCL:
   #_w1 := "DB100_WORK_BIT"."STAT22_Water Pulser" AND NOT "Tag_16";   // rising edge
   "Tag_16" := "DB100_WORK_BIT"."STAT22_Water Pulser";
   IF #_w1 THEN
       "DB102_ANALOG_DISPLAY".STAT24_TOTAL_WATER := "DB102_ANALOG_DISPLAY".STAT24_TOTAL_WATER + 0.1;
   END_IF;
END_REGION

REGION Network 3: RESET TOTAL WATER
   RUNG wire#powerrail
      { S7_Templates := "SrcType := Real" } GT_Contact(in1 := "DB102_ANALOG_DISPLAY".STAT24_TOTAL_WATER, in2 := 999999.9)
      Move(in := 0.0, out1 => "DB102_ANALOG_DISPLAY".STAT24_TOTAL_WATER)
   END_RUNG
   // the same network as SCL:
   IF "DB102_ANALOG_DISPLAY".STAT24_TOTAL_WATER > 999999.9 THEN
       "DB102_ANALOG_DISPLAY".STAT24_TOTAL_WATER := 0.0;
   END_IF;
END_REGION
END_FUNCTION

FUNCTION "FC8_MOTOR_STATUS" : Void   // FC8, LAD
TITLE = HMI STATUS IN DB 154 TO HMI
{ S7_Optimized_Access := 'TRUE' }
VERSION : 0.1
BEGIN

REGION Network 1: HMI STATUS FEED PUMP 1
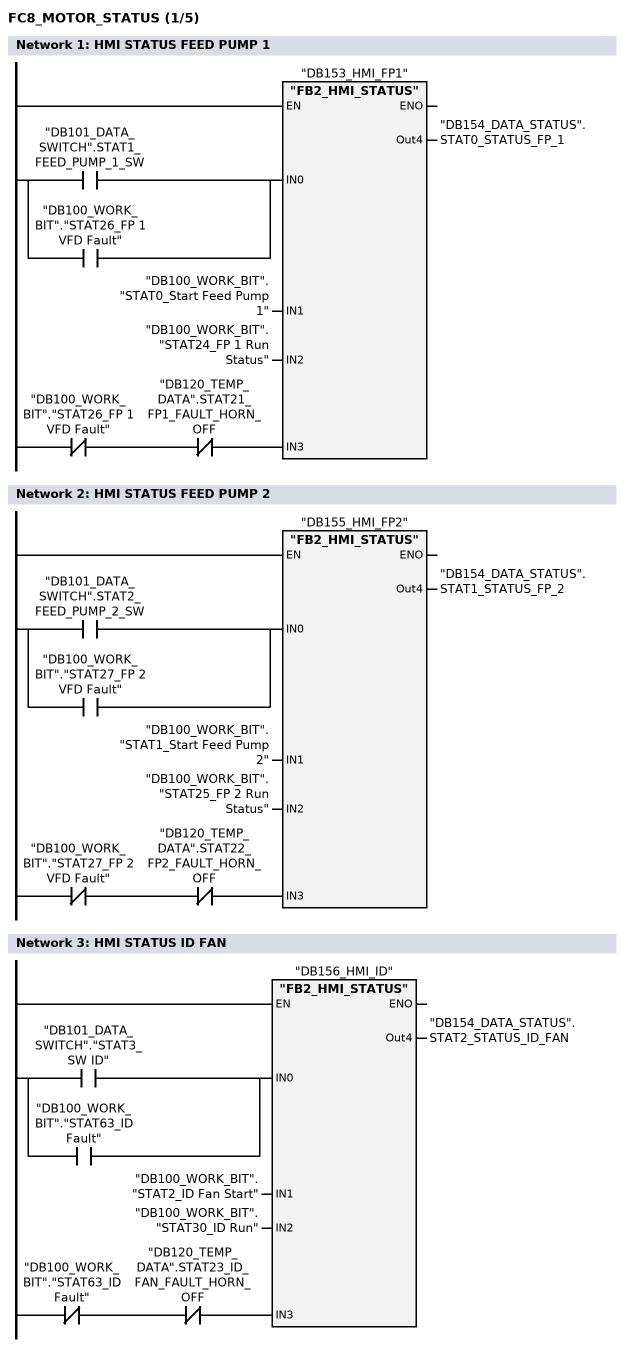
   RUNG wire#powerrail
      "DB153_HMI_FP1"(IN0 := wire#w1, IN3 := wire#w2, IN1 := "DB100_WORK_BIT"."STAT0_Start Feed Pump 1", IN2 := "DB100_WORK_BIT"."STAT24_FP 1 Run Status", Out4 => "DB154_DATA_STATUS".STAT0_STATUS_FP_1)
   END_RUNG
   RUNG wire#powerrail
      Contact( "DB101_DATA_SWITCH".STAT1_FEED_PUMP_1_SW )
   END_RUNG wire#w1
   RUNG wire#powerrail
      Contact( "DB100_WORK_BIT"."STAT26_FP 1 VFD Fault" )
   END_RUNG wire#w1
   RUNG wire#powerrail
      I_Contact( "DB100_WORK_BIT"."STAT26_FP 1 VFD Fault" )
      I_Contact( "DB120_TEMP_DATA".STAT21_FP1_FAULT_HORN_OFF )
   END_RUNG wire#w2
   // the same network as SCL:
   "DB153_HMI_FP1"(IN0 := "DB101_DATA_SWITCH".STAT1_FEED_PUMP_1_SW OR "DB100_WORK_BIT"."STAT26_FP 1 VFD Fault",   // "FB2_HMI_STATUS"
                   IN1 := "DB100_WORK_BIT"."STAT0_Start Feed Pump 1",
                   IN2 := "DB100_WORK_BIT"."STAT24_FP 1 Run Status",
                   IN3 := NOT "DB100_WORK_BIT"."STAT26_FP 1 VFD Fault" AND NOT "DB120_TEMP_DATA".STAT21_FP1_FAULT_HORN_OFF,
                   Out4 => "DB154_DATA_STATUS".STAT0_STATUS_FP_1);
END_REGION

REGION Network 2: HMI STATUS FEED PUMP 2
   RUNG wire#powerrail
      "DB155_HMI_FP2"(IN0 := wire#w1, IN3 := wire#w2, IN1 := "DB100_WORK_BIT"."STAT1_Start Feed Pump 2", IN2 := "DB100_WORK_BIT"."STAT25_FP 2 Run Status", Out4 => "DB154_DATA_STATUS".STAT1_STATUS_FP_2)
   END_RUNG
   RUNG wire#powerrail
      Contact( "DB101_DATA_SWITCH".STAT2_FEED_PUMP_2_SW )
   END_RUNG wire#w1
   RUNG wire#powerrail
      Contact( "DB100_WORK_BIT"."STAT27_FP 2 VFD Fault" )
   END_RUNG wire#w1
   RUNG wire#powerrail
      I_Contact( "DB100_WORK_BIT"."STAT27_FP 2 VFD Fault" )
      I_Contact( "DB120_TEMP_DATA".STAT22_FP2_FAULT_HORN_OFF )
   END_RUNG wire#w2
   // the same network as SCL:
   "DB155_HMI_FP2"(IN0 := "DB101_DATA_SWITCH".STAT2_FEED_PUMP_2_SW OR "DB100_WORK_BIT"."STAT27_FP 2 VFD Fault",   // "FB2_HMI_STATUS"
                   IN1 := "DB100_WORK_BIT"."STAT1_Start Feed Pump 2",
                   IN2 := "DB100_WORK_BIT"."STAT25_FP 2 Run Status",
                   IN3 := NOT "DB100_WORK_BIT"."STAT27_FP 2 VFD Fault" AND NOT "DB120_TEMP_DATA".STAT22_FP2_FAULT_HORN_OFF,
                   Out4 => "DB154_DATA_STATUS".STAT1_STATUS_FP_2);
END_REGION

REGION Network 3: HMI STATUS ID FAN
   RUNG wire#powerrail
      "DB156_HMI_ID"(IN0 := wire#w1, IN3 := wire#w2, IN1 := "DB100_WORK_BIT"."STAT2_ID Fan Start", IN2 := "DB100_WORK_BIT"."STAT30_ID Run", Out4 => "DB154_DATA_STATUS".STAT2_STATUS_ID_FAN)
   END_RUNG
   RUNG wire#powerrail
      Contact( "DB101_DATA_SWITCH"."STAT3_SW ID" )
   END_RUNG wire#w1
   RUNG wire#powerrail
      Contact( "DB100_WORK_BIT"."STAT63_ID Fault" )
   END_RUNG wire#w1
   RUNG wire#powerrail
      I_Contact( "DB100_WORK_BIT"."STAT63_ID Fault" )
      I_Contact( "DB120_TEMP_DATA".STAT23_ID_FAN_FAULT_HORN_OFF )
   END_RUNG wire#w2
   // the same network as SCL:
   "DB156_HMI_ID"(IN0 := "DB101_DATA_SWITCH"."STAT3_SW ID" OR "DB100_WORK_BIT"."STAT63_ID Fault",   // "FB2_HMI_STATUS"
                  IN1 := "DB100_WORK_BIT"."STAT2_ID Fan Start",
                  IN2 := "DB100_WORK_BIT"."STAT30_ID Run",
                  IN3 := NOT "DB100_WORK_BIT"."STAT63_ID Fault" AND NOT "DB120_TEMP_DATA".STAT23_ID_FAN_FAULT_HORN_OFF,
                  Out4 => "DB154_DATA_STATUS".STAT2_STATUS_ID_FAN);
END_REGION

REGION Network 4: HMI STATUS LH FD FAN
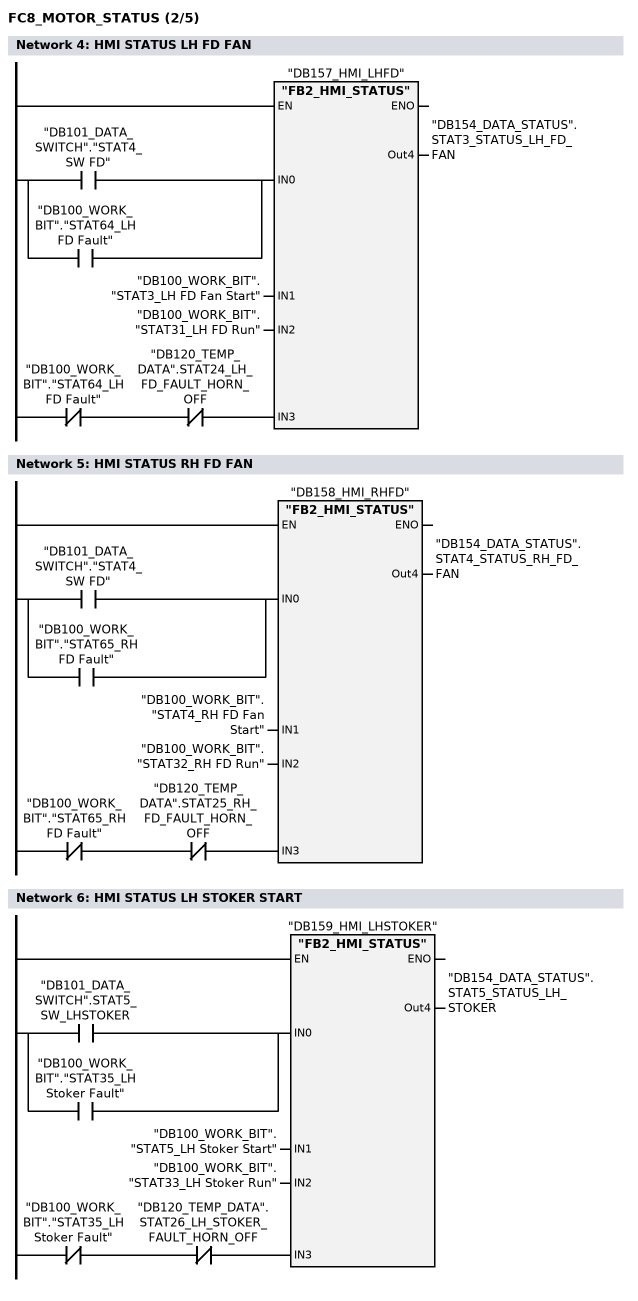
   RUNG wire#powerrail
      "DB157_HMI_LHFD"(IN0 := wire#w1, IN3 := wire#w2, IN1 := "DB100_WORK_BIT"."STAT3_LH FD Fan Start", IN2 := "DB100_WORK_BIT"."STAT31_LH FD Run", Out4 => "DB154_DATA_STATUS".STAT3_STATUS_LH_FD_FAN)
   END_RUNG
   RUNG wire#powerrail
      Contact( "DB101_DATA_SWITCH"."STAT4_SW FD" )
   END_RUNG wire#w1
   RUNG wire#powerrail
      Contact( "DB100_WORK_BIT"."STAT64_LH FD Fault" )
   END_RUNG wire#w1
   RUNG wire#powerrail
      I_Contact( "DB100_WORK_BIT"."STAT64_LH FD Fault" )
      I_Contact( "DB120_TEMP_DATA".STAT24_LH_FD_FAULT_HORN_OFF )
   END_RUNG wire#w2
   // the same network as SCL:
   "DB157_HMI_LHFD"(IN0 := "DB101_DATA_SWITCH"."STAT4_SW FD" OR "DB100_WORK_BIT"."STAT64_LH FD Fault",   // "FB2_HMI_STATUS"
                    IN1 := "DB100_WORK_BIT"."STAT3_LH FD Fan Start",
                    IN2 := "DB100_WORK_BIT"."STAT31_LH FD Run",
                    IN3 := NOT "DB100_WORK_BIT"."STAT64_LH FD Fault" AND NOT "DB120_TEMP_DATA".STAT24_LH_FD_FAULT_HORN_OFF,
                    Out4 => "DB154_DATA_STATUS".STAT3_STATUS_LH_FD_FAN);
END_REGION

REGION Network 5: HMI STATUS RH FD FAN
   RUNG wire#powerrail
      "DB158_HMI_RHFD"(IN0 := wire#w1, IN3 := wire#w2, IN1 := "DB100_WORK_BIT"."STAT4_RH FD Fan Start", IN2 := "DB100_WORK_BIT"."STAT32_RH FD Run", Out4 => "DB154_DATA_STATUS".STAT4_STATUS_RH_FD_FAN)
   END_RUNG
   RUNG wire#powerrail
      Contact( "DB101_DATA_SWITCH"."STAT4_SW FD" )
   END_RUNG wire#w1
   RUNG wire#powerrail
      Contact( "DB100_WORK_BIT"."STAT65_RH FD Fault" )
   END_RUNG wire#w1
   RUNG wire#powerrail
      I_Contact( "DB100_WORK_BIT"."STAT65_RH FD Fault" )
      I_Contact( "DB120_TEMP_DATA".STAT25_RH_FD_FAULT_HORN_OFF )
   END_RUNG wire#w2
   // the same network as SCL:
   "DB158_HMI_RHFD"(IN0 := "DB101_DATA_SWITCH"."STAT4_SW FD" OR "DB100_WORK_BIT"."STAT65_RH FD Fault",   // "FB2_HMI_STATUS"
                    IN1 := "DB100_WORK_BIT"."STAT4_RH FD Fan Start",
                    IN2 := "DB100_WORK_BIT"."STAT32_RH FD Run",
                    IN3 := NOT "DB100_WORK_BIT"."STAT65_RH FD Fault" AND NOT "DB120_TEMP_DATA".STAT25_RH_FD_FAULT_HORN_OFF,
                    Out4 => "DB154_DATA_STATUS".STAT4_STATUS_RH_FD_FAN);
END_REGION

REGION Network 6: HMI STATUS LH STOKER START
   RUNG wire#powerrail
      "DB159_HMI_LHSTOKER"(IN0 := wire#w1, IN3 := wire#w2, IN1 := "DB100_WORK_BIT"."STAT5_LH Stoker Start", IN2 := "DB100_WORK_BIT"."STAT33_LH Stoker Run", Out4 => "DB154_DATA_STATUS".STAT5_STATUS_LH_STOKER)
   END_RUNG
   RUNG wire#powerrail
      Contact( "DB101_DATA_SWITCH".STAT5_SW_LHSTOKER )
   END_RUNG wire#w1
   RUNG wire#powerrail
      Contact( "DB100_WORK_BIT"."STAT35_LH Stoker Fault" )
   END_RUNG wire#w1
   RUNG wire#powerrail
      I_Contact( "DB100_WORK_BIT"."STAT35_LH Stoker Fault" )
      I_Contact( "DB120_TEMP_DATA".STAT26_LH_STOKER_FAULT_HORN_OFF )
   END_RUNG wire#w2
   // the same network as SCL:
   "DB159_HMI_LHSTOKER"(IN0 := "DB101_DATA_SWITCH".STAT5_SW_LHSTOKER OR "DB100_WORK_BIT"."STAT35_LH Stoker Fault",   // "FB2_HMI_STATUS"
                        IN1 := "DB100_WORK_BIT"."STAT5_LH Stoker Start",
                        IN2 := "DB100_WORK_BIT"."STAT33_LH Stoker Run",
                        IN3 := NOT "DB100_WORK_BIT"."STAT35_LH Stoker Fault" AND NOT "DB120_TEMP_DATA".STAT26_LH_STOKER_FAULT_HORN_OFF,
                        Out4 => "DB154_DATA_STATUS".STAT5_STATUS_LH_STOKER);
END_REGION

REGION Network 7: HMI STATUS RH STOKER START
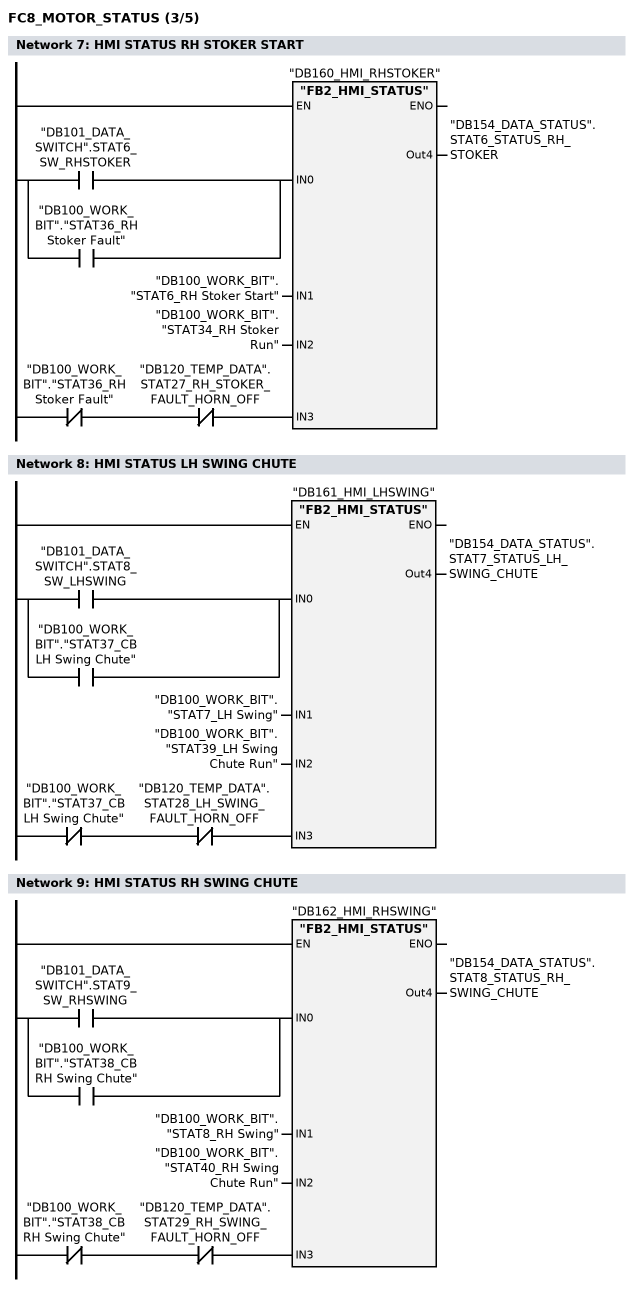
   RUNG wire#powerrail
      "DB160_HMI_RHSTOKER"(IN0 := wire#w1, IN3 := wire#w2, IN1 := "DB100_WORK_BIT"."STAT6_RH Stoker Start", IN2 := "DB100_WORK_BIT"."STAT34_RH Stoker Run", Out4 => "DB154_DATA_STATUS".STAT6_STATUS_RH_STOKER)
   END_RUNG
   RUNG wire#powerrail
      Contact( "DB101_DATA_SWITCH".STAT6_SW_RHSTOKER )
   END_RUNG wire#w1
   RUNG wire#powerrail
      Contact( "DB100_WORK_BIT"."STAT36_RH Stoker Fault" )
   END_RUNG wire#w1
   RUNG wire#powerrail
      I_Contact( "DB100_WORK_BIT"."STAT36_RH Stoker Fault" )
      I_Contact( "DB120_TEMP_DATA".STAT27_RH_STOKER_FAULT_HORN_OFF )
   END_RUNG wire#w2
   // the same network as SCL:
   "DB160_HMI_RHSTOKER"(IN0 := "DB101_DATA_SWITCH".STAT6_SW_RHSTOKER OR "DB100_WORK_BIT"."STAT36_RH Stoker Fault",   // "FB2_HMI_STATUS"
                        IN1 := "DB100_WORK_BIT"."STAT6_RH Stoker Start",
                        IN2 := "DB100_WORK_BIT"."STAT34_RH Stoker Run",
                        IN3 := NOT "DB100_WORK_BIT"."STAT36_RH Stoker Fault" AND NOT "DB120_TEMP_DATA".STAT27_RH_STOKER_FAULT_HORN_OFF,
                        Out4 => "DB154_DATA_STATUS".STAT6_STATUS_RH_STOKER);
END_REGION

REGION Network 8: HMI STATUS LH SWING CHUTE
   RUNG wire#powerrail
      "DB161_HMI_LHSWING"(IN0 := wire#w1, IN3 := wire#w2, IN1 := "DB100_WORK_BIT"."STAT7_LH Swing", IN2 := "DB100_WORK_BIT"."STAT39_LH Swing Chute Run", Out4 => "DB154_DATA_STATUS".STAT7_STATUS_LH_SWING_CHUTE)
   END_RUNG
   RUNG wire#powerrail
      Contact( "DB101_DATA_SWITCH".STAT8_SW_LHSWING )
   END_RUNG wire#w1
   RUNG wire#powerrail
      Contact( "DB100_WORK_BIT"."STAT37_CB LH Swing Chute" )
   END_RUNG wire#w1
   RUNG wire#powerrail
      I_Contact( "DB100_WORK_BIT"."STAT37_CB LH Swing Chute" )
      I_Contact( "DB120_TEMP_DATA".STAT28_LH_SWING_FAULT_HORN_OFF )
   END_RUNG wire#w2
   // the same network as SCL:
   "DB161_HMI_LHSWING"(IN0 := "DB101_DATA_SWITCH".STAT8_SW_LHSWING OR "DB100_WORK_BIT"."STAT37_CB LH Swing Chute",   // "FB2_HMI_STATUS"
                       IN1 := "DB100_WORK_BIT"."STAT7_LH Swing",
                       IN2 := "DB100_WORK_BIT"."STAT39_LH Swing Chute Run",
                       IN3 := NOT "DB100_WORK_BIT"."STAT37_CB LH Swing Chute" AND NOT "DB120_TEMP_DATA".STAT28_LH_SWING_FAULT_HORN_OFF,
                       Out4 => "DB154_DATA_STATUS".STAT7_STATUS_LH_SWING_CHUTE);
END_REGION

REGION Network 9: HMI STATUS RH SWING CHUTE
   RUNG wire#powerrail
      "DB162_HMI_RHSWING"(IN0 := wire#w1, IN3 := wire#w2, IN1 := "DB100_WORK_BIT"."STAT8_RH Swing", IN2 := "DB100_WORK_BIT"."STAT40_RH Swing Chute Run", Out4 => "DB154_DATA_STATUS".STAT8_STATUS_RH_SWING_CHUTE)
   END_RUNG
   RUNG wire#powerrail
      Contact( "DB101_DATA_SWITCH".STAT9_SW_RHSWING )
   END_RUNG wire#w1
   RUNG wire#powerrail
      Contact( "DB100_WORK_BIT"."STAT38_CB RH Swing Chute" )
   END_RUNG wire#w1
   RUNG wire#powerrail
      I_Contact( "DB100_WORK_BIT"."STAT38_CB RH Swing Chute" )
      I_Contact( "DB120_TEMP_DATA".STAT29_RH_SWING_FAULT_HORN_OFF )
   END_RUNG wire#w2
   // the same network as SCL:
   "DB162_HMI_RHSWING"(IN0 := "DB101_DATA_SWITCH".STAT9_SW_RHSWING OR "DB100_WORK_BIT"."STAT38_CB RH Swing Chute",   // "FB2_HMI_STATUS"
                       IN1 := "DB100_WORK_BIT"."STAT8_RH Swing",
                       IN2 := "DB100_WORK_BIT"."STAT40_RH Swing Chute Run",
                       IN3 := NOT "DB100_WORK_BIT"."STAT38_CB RH Swing Chute" AND NOT "DB120_TEMP_DATA".STAT29_RH_SWING_FAULT_HORN_OFF,
                       Out4 => "DB154_DATA_STATUS".STAT8_STATUS_RH_SWING_CHUTE);
END_REGION

REGION Network 10: HMI STATUS ASH CONVEYOR
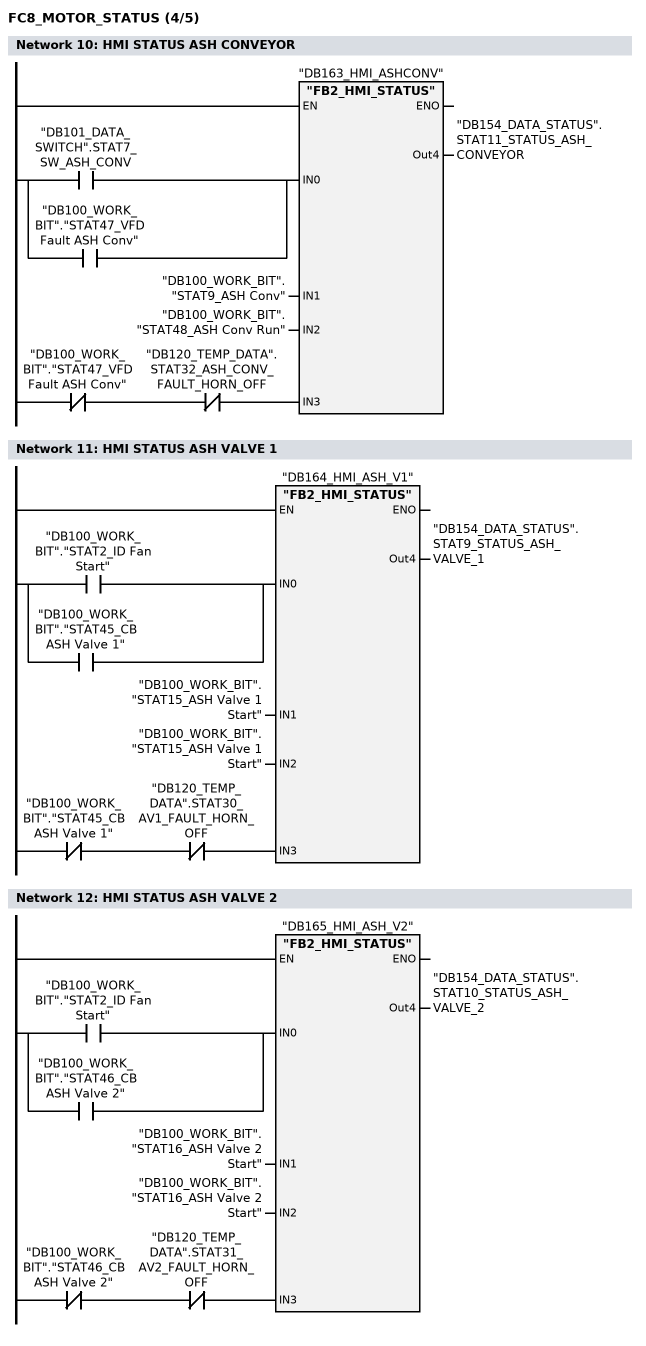
   RUNG wire#powerrail
      "DB163_HMI_ASHCONV"(IN0 := wire#w1, IN3 := wire#w2, IN1 := "DB100_WORK_BIT"."STAT9_ASH Conv", IN2 := "DB100_WORK_BIT"."STAT48_ASH Conv Run", Out4 => "DB154_DATA_STATUS".STAT11_STATUS_ASH_CONVEYOR)
   END_RUNG
   RUNG wire#powerrail
      Contact( "DB101_DATA_SWITCH".STAT7_SW_ASH_CONV )
   END_RUNG wire#w1
   RUNG wire#powerrail
      Contact( "DB100_WORK_BIT"."STAT47_VFD Fault ASH Conv" )
   END_RUNG wire#w1
   RUNG wire#powerrail
      I_Contact( "DB100_WORK_BIT"."STAT47_VFD Fault ASH Conv" )
      I_Contact( "DB120_TEMP_DATA".STAT32_ASH_CONV_FAULT_HORN_OFF )
   END_RUNG wire#w2
   // the same network as SCL:
   "DB163_HMI_ASHCONV"(IN0 := "DB101_DATA_SWITCH".STAT7_SW_ASH_CONV OR "DB100_WORK_BIT"."STAT47_VFD Fault ASH Conv",   // "FB2_HMI_STATUS"
                       IN1 := "DB100_WORK_BIT"."STAT9_ASH Conv",
                       IN2 := "DB100_WORK_BIT"."STAT48_ASH Conv Run",
                       IN3 := NOT "DB100_WORK_BIT"."STAT47_VFD Fault ASH Conv" AND NOT "DB120_TEMP_DATA".STAT32_ASH_CONV_FAULT_HORN_OFF,
                       Out4 => "DB154_DATA_STATUS".STAT11_STATUS_ASH_CONVEYOR);
END_REGION

REGION Network 11: HMI STATUS ASH VALVE 1
   RUNG wire#powerrail
      "DB164_HMI_ASH_V1"(IN0 := wire#w1, IN3 := wire#w2, IN1 := "DB100_WORK_BIT"."STAT15_ASH Valve 1 Start", IN2 := "DB100_WORK_BIT"."STAT15_ASH Valve 1 Start", Out4 => "DB154_DATA_STATUS".STAT9_STATUS_ASH_VALVE_1)
   END_RUNG
   RUNG wire#powerrail
      Contact( "DB100_WORK_BIT"."STAT2_ID Fan Start" )
   END_RUNG wire#w1
   RUNG wire#powerrail
      Contact( "DB100_WORK_BIT"."STAT45_CB ASH Valve 1" )
   END_RUNG wire#w1
   RUNG wire#powerrail
      I_Contact( "DB100_WORK_BIT"."STAT45_CB ASH Valve 1" )
      I_Contact( "DB120_TEMP_DATA".STAT30_AV1_FAULT_HORN_OFF )
   END_RUNG wire#w2
   // the same network as SCL:
   "DB164_HMI_ASH_V1"(IN0 := "DB100_WORK_BIT"."STAT2_ID Fan Start" OR "DB100_WORK_BIT"."STAT45_CB ASH Valve 1",   // "FB2_HMI_STATUS"
                      IN1 := "DB100_WORK_BIT"."STAT15_ASH Valve 1 Start",
                      IN2 := "DB100_WORK_BIT"."STAT15_ASH Valve 1 Start",
                      IN3 := NOT "DB100_WORK_BIT"."STAT45_CB ASH Valve 1" AND NOT "DB120_TEMP_DATA".STAT30_AV1_FAULT_HORN_OFF,
                      Out4 => "DB154_DATA_STATUS".STAT9_STATUS_ASH_VALVE_1);
END_REGION

REGION Network 12: HMI STATUS ASH VALVE 2
   RUNG wire#powerrail
      "DB165_HMI_ASH_V2"(IN0 := wire#w1, IN3 := wire#w2, IN1 := "DB100_WORK_BIT"."STAT16_ASH Valve 2 Start", IN2 := "DB100_WORK_BIT"."STAT16_ASH Valve 2 Start", Out4 => "DB154_DATA_STATUS".STAT10_STATUS_ASH_VALVE_2)
   END_RUNG
   RUNG wire#powerrail
      Contact( "DB100_WORK_BIT"."STAT2_ID Fan Start" )
   END_RUNG wire#w1
   RUNG wire#powerrail
      Contact( "DB100_WORK_BIT"."STAT46_CB ASH Valve 2" )
   END_RUNG wire#w1
   RUNG wire#powerrail
      I_Contact( "DB100_WORK_BIT"."STAT46_CB ASH Valve 2" )
      I_Contact( "DB120_TEMP_DATA".STAT31_AV2_FAULT_HORN_OFF )
   END_RUNG wire#w2
   // the same network as SCL:
   "DB165_HMI_ASH_V2"(IN0 := "DB100_WORK_BIT"."STAT2_ID Fan Start" OR "DB100_WORK_BIT"."STAT46_CB ASH Valve 2",   // "FB2_HMI_STATUS"
                      IN1 := "DB100_WORK_BIT"."STAT16_ASH Valve 2 Start",
                      IN2 := "DB100_WORK_BIT"."STAT16_ASH Valve 2 Start",
                      IN3 := NOT "DB100_WORK_BIT"."STAT46_CB ASH Valve 2" AND NOT "DB120_TEMP_DATA".STAT31_AV2_FAULT_HORN_OFF,
                      Out4 => "DB154_DATA_STATUS".STAT10_STATUS_ASH_VALVE_2);
END_REGION

REGION Network 13: HMI STATUS WETSCRUBBER
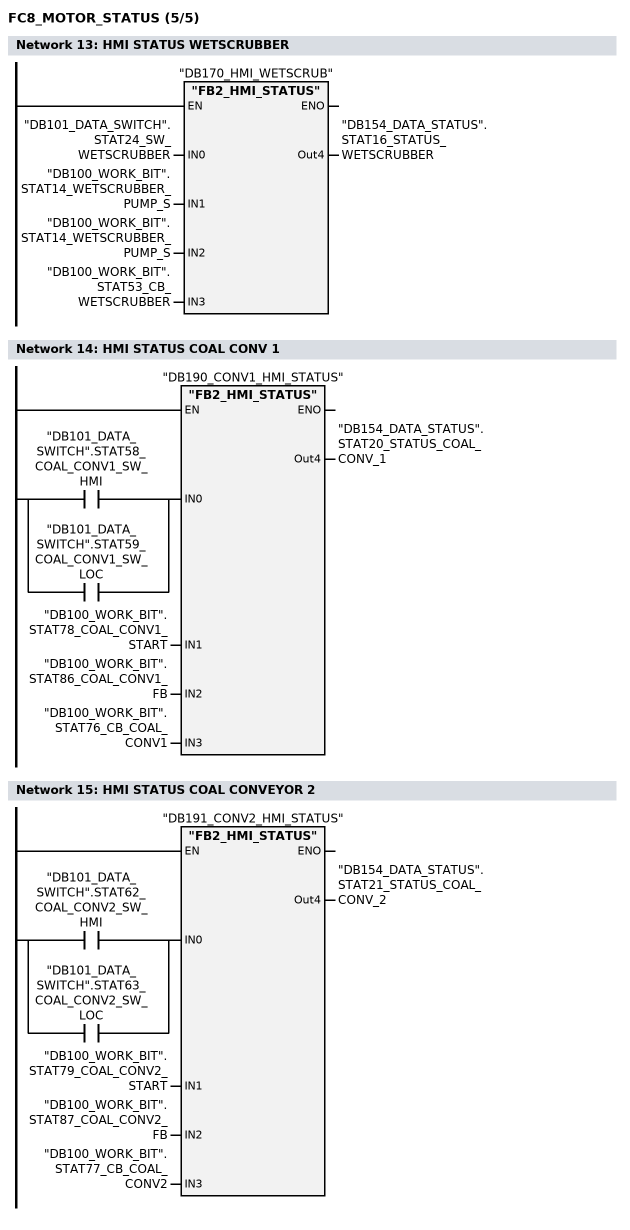
   RUNG wire#powerrail
      "DB170_HMI_WETSCRUB"(IN0 := "DB101_DATA_SWITCH".STAT24_SW_WETSCRUBBER, IN1 := "DB100_WORK_BIT".STAT14_WETSCRUBBER_PUMP_S, IN2 := "DB100_WORK_BIT".STAT14_WETSCRUBBER_PUMP_S, IN3 := "DB100_WORK_BIT".STAT53_CB_WETSCRUBBER, Out4 => "DB154_DATA_STATUS".STAT16_STATUS_WETSCRUBBER)
   END_RUNG
   // the same network as SCL:
   "DB170_HMI_WETSCRUB"(IN0 := "DB101_DATA_SWITCH".STAT24_SW_WETSCRUBBER,   // "FB2_HMI_STATUS"
                        IN1 := "DB100_WORK_BIT".STAT14_WETSCRUBBER_PUMP_S,
                        IN2 := "DB100_WORK_BIT".STAT14_WETSCRUBBER_PUMP_S,
                        IN3 := "DB100_WORK_BIT".STAT53_CB_WETSCRUBBER,
                        Out4 => "DB154_DATA_STATUS".STAT16_STATUS_WETSCRUBBER);
END_REGION

REGION Network 14: HMI STATUS COAL CONV 1
   RUNG wire#powerrail
      "DB190_CONV1_HMI_STATUS"(IN0 := wire#w1, IN1 := "DB100_WORK_BIT".STAT78_COAL_CONV1_START, IN2 := "DB100_WORK_BIT".STAT86_COAL_CONV1_FB, IN3 := "DB100_WORK_BIT".STAT76_CB_COAL_CONV1, Out4 => "DB154_DATA_STATUS".STAT20_STATUS_COAL_CONV_1)
   END_RUNG
   RUNG wire#powerrail
      Contact( "DB101_DATA_SWITCH".STAT58_COAL_CONV1_SW_HMI )
   END_RUNG wire#w1
   RUNG wire#powerrail
      Contact( "DB101_DATA_SWITCH".STAT59_COAL_CONV1_SW_LOC )
   END_RUNG wire#w1
   // the same network as SCL:
   "DB190_CONV1_HMI_STATUS"(IN0 := "DB101_DATA_SWITCH".STAT58_COAL_CONV1_SW_HMI OR "DB101_DATA_SWITCH".STAT59_COAL_CONV1_SW_LOC,   // "FB2_HMI_STATUS"
                           IN1 := "DB100_WORK_BIT".STAT78_COAL_CONV1_START,
                           IN2 := "DB100_WORK_BIT".STAT86_COAL_CONV1_FB,
                           IN3 := "DB100_WORK_BIT".STAT76_CB_COAL_CONV1,
                           Out4 => "DB154_DATA_STATUS".STAT20_STATUS_COAL_CONV_1);
END_REGION

REGION Network 15: HMI STATUS COAL CONVEYOR 2
   RUNG wire#powerrail
      "DB191_CONV2_HMI_STATUS"(IN0 := wire#w1, IN1 := "DB100_WORK_BIT".STAT79_COAL_CONV2_START, IN2 := "DB100_WORK_BIT".STAT87_COAL_CONV2_FB, IN3 := "DB100_WORK_BIT".STAT77_CB_COAL_CONV2, Out4 => "DB154_DATA_STATUS".STAT21_STATUS_COAL_CONV_2)
   END_RUNG
   RUNG wire#powerrail
      Contact( "DB101_DATA_SWITCH".STAT62_COAL_CONV2_SW_HMI )
   END_RUNG wire#w1
   RUNG wire#powerrail
      Contact( "DB101_DATA_SWITCH".STAT63_COAL_CONV2_SW_LOC )
   END_RUNG wire#w1
   // the same network as SCL:
   "DB191_CONV2_HMI_STATUS"(IN0 := "DB101_DATA_SWITCH".STAT62_COAL_CONV2_SW_HMI OR "DB101_DATA_SWITCH".STAT63_COAL_CONV2_SW_LOC,   // "FB2_HMI_STATUS"
                           IN1 := "DB100_WORK_BIT".STAT79_COAL_CONV2_START,
                           IN2 := "DB100_WORK_BIT".STAT87_COAL_CONV2_FB,
                           IN3 := "DB100_WORK_BIT".STAT77_CB_COAL_CONV2,
                           Out4 => "DB154_DATA_STATUS".STAT21_STATUS_COAL_CONV_2);
END_REGION
END_FUNCTION

FUNCTION "FC9_Undergrate_Damper" : Void   // FC9, LAD
TITLE = UNDER GRATE DAMPER
{ S7_Optimized_Access := 'TRUE' }
VERSION : 0.1
// SPEED LH FD FAN = IW 112
// SPEED RH FD FAN = IW 114
// 
// DIGITAL OUTPUT LH FRONT OPEN = Q4.4
// DIGITAL OUTPUT LH FRONT CLOSE = Q4.5
// 
// DIGITAL OUTPUT RH FRONT OPEN = Q4.6
// DIGITAL OUTPUT RH FRONT CLOSE = Q4.7
// 
// DIGITAL OUTPUT LH REAR OPEN = Q5.0
// DIGITAL OUTPUT LH REAR CLOSE = Q5.1
// 
// DIGITAL OUTPUT RH REAR OPEN = Q5.2
// DIGITAL OUTPUT RH REAR CLOSE = Q5.3
   VAR_TEMP   // added for the SCL form of the ladder/FBD networks
      _w1 : Bool;
   END_VAR
BEGIN

REGION Network 1: SCALLING Speed LH FD Fan | IW 112
